LIN {X 0,Y 416.989,Z 554.741,A -85,B 0,C 180,E1 -10166.135,E2 -10166.135} C_VEL
LIN {X 0,Y 417.027,Z 556.75,A -85,B 0,C 180,E1 -10168.069,E2 -10168.069} C_VEL
LIN {X 0,Y 416.981,Z 557.414,A -85,B 0,C 180,E1 -10170,E2 -10170} C_VEL
LIN {X 0,Y 417.027,Z 556.748,A -85,B 0,C 180,E1 -10171.932,E2 -10171.932} C_VEL
LIN {X 0,Y 416.989,Z 554.738,A -85,B 0,C 180,E1 -10173.866,E2 -10173.866} C_VEL
LIN {X 0,Y 417.129,Z 551.337,A -85,B 0,C 180,E1 -10175.802,E2 -10175.802} C_VEL
LIN {X 0,Y 417.316,Z 546.442,A -85,B 0,C 180,E1 -10177.743,E2 -10177.743} C_VEL
LIN {X 0,Y 417.74,Z 539.91,A -85,B 0,C 180,E1 -10179.685,E2 -10179.685} C_VEL
LIN {X 0,Y 418.314,Z 532.641,A -85,B 0,C 180,E1 -10181.385,E2 -10181.385} C_VEL
LIN {X 0,Y 418.978,Z 524.176,A -85,B 0,C 180,E1 -10182.995,E2 -10182.995} C_VEL
LIN {X 0,Y 419.845,Z 514.188,A -85,B 0,C 180,E1 -10184.542,E2 -10184.542} C_VEL
LIN {X 0,Y 420.766,Z 503.727,A -85,B 0,C 180,E1 -10185.873,E2 -10185.873} C_VEL
LIN {X 0,Y 421.802,Z 492.183,A -85,B 0,C 180,E1 -10187.077,E2 -10187.077} C_VEL
LIN {X 0,Y 422.858,Z 479.374,A -85,B 0,C 180,E1 -10188.157,E2 -10188.157} C_VEL
LIN {X 0,Y 423.8,Z 466.334,A -85,B 0,C 180,E1 -10189.025,E2 -10189.025} C_VEL
LIN {X 0,Y 424.522,Z 452.931,A -85,B 0,C 180,E1 -10189.713,E2 -10189.713} C_VEL
LIN {X 0,Y 425.232,Z 438.211,A -85,B 0,C 180,E1 -10190.245,E2 -10190.245} C_VEL
LIN {X 0,Y 425.645,Z 423.401,A -85,B 0,C 180,E1 -10190.572,E2 -10190.572} C_VEL
LIN {X 0,Y 426.978,Z 321.763,A -85,B 0,C 180,E1 -10192.302,E2 -10192.302} C_VEL
LIN {X 0,Y 421.78,Z 294.783,A -85,B 0,C 180,E1 -10193.108,E2 -10193.108} C_VEL
LIN {X 0,Y 422.402,Z 285.458,A -85,B 0,C 180,E1 -10194.841,E2 -10194.841} C_VEL
LIN {X 0,Y 420.106,Z 273.797,A -85,B 0,C 180,E1 -10197.302,E2 -10197.302} C_VEL
LIN {X 0,Y 418.323,Z 266.179,A -85,B 0,C 180,E1 -10199.01,E2 -10199.01} C_VEL
LIN {X 0,Y 418.244,Z 266.011,A -85,B 0,C 180,E1 -10202.527,E2 -10202.527} C_VEL
LIN {X 0,Y 418.257,Z 266.012,A -85,B 0,C 180,E1 -10204.84,E2 -10204.84} C_VEL
LIN {X 0,Y 418.25,Z 266.009,A -85,B 0,C 180,E1 -10208.441,E2 -10208.441} C_VEL
LIN {X 0,Y 418.219,Z 265.999,A -85,B 0,C 180,E1 -10210.947,E2 -10210.947} C_VEL
LIN {X 0,Y 418.213,Z 266.013,A -85,B 0,C 180,E1 -10213.73,E2 -10213.73} C_VEL
LIN {X 0,Y 418.205,Z 266.016,A -85,B 0,C 180,E1 -10216.448,E2 -10216.448} C_VEL
LIN {X 0,Y 418.22,Z 266.007,A -85,B 0,C 180,E1 -10219.129,E2 -10219.129} C_VEL
LIN {X 0,Y 418.23,Z 266.013,A -85,B 0,C 180,E1 -10222.165,E2 -10222.165} C_VEL
LIN {X 0,Y 418.26,Z 265.977,A -85,B 0,C 180,E1 -10225.419,E2 -10225.419} C_VEL
LIN {X 0,Y 418.217,Z 266.013,A -85,B 0,C 180,E1 -10228.604,E2 -10228.604} C_VEL
LIN {X 0,Y 418.289,Z 266,A -85,B 0,C 180,E1 -10231.937,E2 -10231.937} C_VEL
LIN {X 0,Y 418.283,Z 266.004,A -85,B 0,C 180,E1 -10235.162,E2 -10235.162} C_VEL
LIN {X 0,Y 418.227,Z 266.008,A -85,B 0,C 180,E1 -10238.303,E2 -10238.303} C_VEL
LIN {X 0,Y 418.276,Z 266.007,A -85,B 0,C 180,E1 -10241.383,E2 -10241.383} C_VEL
LIN {X 0,Y 418.294,Z 266,A -85,B 0,C 180,E1 -10244.406,E2 -10244.406} C_VEL
LIN {X 0,Y 418.348,Z 265.999,A -85,B 0,C 180,E1 -10247.385,E2 -10247.385} C_VEL
LIN {X 0,Y 418.333,Z 265.992,A -85,B 0,C 180,E1 -10250.329,E2 -10250.329} C_VEL
LIN {X 0,Y 418.506,Z 265.977,A -85,B 0,C 180,E1 -10252.279,E2 -10252.279} C_VEL
LIN {X 0,Y 418.505,Z 265.972,A -85,B 0,C 180,E1 -10254.217,E2 -10254.217} C_VEL
LIN {X 0,Y 418.537,Z 265.973,A -85,B 0,C 180,E1 -10258.076,E2 -10258.076} C_VEL
LIN {X 0,Y 418.664,Z 265.956,A -85,B 0,C 180,E1 -10260,E2 -10260} C_VEL
LIN {X 0,Y 418.504,Z 265.964,A -85,B 0,C 180,E1 -10262.888,E2 -10262.888} C_VEL
LIN {X 0,Y 418.486,Z 265.979,A -85,B 0,C 180,E1 -10266.751,E2 -10266.751} C_VEL
LIN {X 0,Y 418.333,Z 265.994,A -85,B 0,C 180,E1 -10269.672,E2 -10269.672} C_VEL
LIN {X 0,Y 418.339,Z 266.001,A -85,B 0,C 180,E1 -10273.001,E2 -10273.001} C_VEL
LIN {X 0,Y 418.306,Z 265.999,A -85,B 0,C 180,E1 -10276.736,E2 -10276.736} C_VEL
LIN {X 0,Y 418.264,Z 266.001,A -85,B 0,C 180,E1 -10279.791,E2 -10279.791} C_VEL
LIN {X 0,Y 418.232,Z 266.01,A -85,B 0,C 180,E1 -10282.737,E2 -10282.737} C_VEL
LIN {X 0,Y 418.264,Z 265.998,A -85,B 0,C 180,E1 -10285.905,E2 -10285.905} C_VEL
LIN {X 0,Y 418.269,Z 266.009,A -85,B 0,C 180,E1 -10289.162,E2 -10289.162} C_VEL
LIN {X 0,Y 418.252,Z 265.98,A -85,B 0,C 180,E1 -10292.845,E2 -10292.845} C_VEL
LIN {X 0,Y 418.244,Z 266.004,A -85,B 0,C 180,E1 -10296.239,E2 -10296.239} C_VEL
LIN {X 0,Y 418.26,Z 266,A -85,B 0,C 180,E1 -10299.681,E2 -10299.681} C_VEL
LIN {X 0,Y 418.241,Z 265.99,A -85,B 0,C 180,E1 -10302.324,E2 -10302.324} C_VEL
LIN {X 0,Y 418.236,Z 266.012,A -85,B 0,C 180,E1 -10305.11,E2 -10305.11} C_VEL
LIN {X 0,Y 418.239,Z 265.993,A -85,B 0,C 180,E1 -10307.768,E2 -10307.768} C_VEL
LIN {X 0,Y 418.256,Z 266.011,A -85,B 0,C 180,E1 -10310.619,E2 -10310.619} C_VEL
LIN {X 0,Y 418.242,Z 266.011,A -85,B 0,C 180,E1 -10313.977,E2 -10313.977} C_VEL
LIN {X 0,Y 418.257,Z 266.011,A -85,B 0,C 180,E1 -10317.157,E2 -10317.157} C_VEL
LIN {X 0,Y 418.268,Z 265.996,A -85,B 0,C 180,E1 -10320.896,E2 -10320.896} C_VEL
LIN {X 0,Y 418.345,Z 266.202,A -85,B 0,C 180,E1 -10322.251,E2 -10322.251} C_VEL
LIN {X 0,Y 420.857,Z 277.948,A -85,B 0,C 180,E1 -10324.922,E2 -10324.922} C_VEL
LIN {X 0,Y 422.1,Z 284.986,A -85,B 0,C 180,E1 -10326.447,E2 -10326.447} C_VEL
LIN {X 0,Y 421.937,Z 287.927,A -85,B 0,C 180,E1 -10326.964,E2 -10326.964} C_VEL
LIN {X 0,Y 427.164,Z 313.752,A -85,B 0,C 180,E1 -10327.742,E2 -10327.742} C_VEL
LIN {X 0,Y 425.741,Z 409.801,A -85,B 0,C 180,E1 -10329.37,E2 -10329.37} C_VEL
LIN {X 0,Y 425.346,Z 427.971,A -85,B 0,C 180,E1 -10329.729,E2 -10329.729} C_VEL
LIN {X 0,Y 424.78,Z 442.274,A -85,B 0,C 180,E1 -10330.205,E2 -10330.205} C_VEL
LIN {X 0,Y 424.143,Z 455.506,A -85,B 0,C 180,E1 -10330.837,E2 -10330.837} C_VEL
LIN {X 0,Y 423.336,Z 467.967,A -85,B 0,C 180,E1 -10331.614,E2 -10331.614} C_VEL
LIN {X 0,Y 422.393,Z 480.205,A -85,B 0,C 180,E1 -10332.573,E2 -10332.573} C_VEL
LIN {X 0,Y 421.296,Z 492.545,A -85,B 0,C 180,E1 -10333.775,E2 -10333.775} C_VEL
LIN {X 0,Y 420.401,Z 502.683,A -85,B 0,C 180,E1 -10334.982,E2 -10334.982} C_VEL
LIN {X 0,Y 419.457,Z 512.747,A -85,B 0,C 180,E1 -10336.434,E2 -10336.434} C_VEL
LIN {X 0,Y 419.259,Z 516.218,A -85,B 0,C 180,E1 -10337.009,E2 -10337.009} C_VEL
LIN {X 0,Y 418.347,Z 519.856,A -85,B 0,C 180,E1 -10337.639,E2 -10337.639} C_VEL
LIN {X 0,Y 415.001,Z 525.435,A -85,B 0,C 180,E1 -10338.669,E2 -10338.669} C_VEL
LIN {X 0,Y 411.657,Z 530.499,A -85,B 0,C 180,E1 -10339.758,E2 -10339.758} C_VEL
LIN {X 0,Y 410.76,Z 533.265,A -85,B 0,C 180,E1 -10340.473,E2 -10340.473} C_VEL
LIN {X 0,Y 410.371,Z 538.623,A -85,B 0,C 180,E1 -10342.125,E2 -10342.125} C_VEL
LIN {X 0,Y 410.13,Z 543.523,A -85,B 0,C 180,E1 -10344.099,E2 -10344.099} C_VEL
LIN {X 0,Y 409.943,Z 546.935,A -85,B 0,C 180,E1 -10346.068,E2 -10346.068} C_VEL
LIN {X 0,Y 409.966,Z 548.961,A -85,B 0,C 180,E1 -10348.035,E2 -10348.035} C_VEL
LIN {X 0,Y 409.905,Z 549.659,A -85,B 0,C 180,E1 -10350,E2 -10350} C_VEL
LIN {X 0,Y 409.966,Z 549.033,A -85,B 0,C 180,E1 -10351.965,E2 -10351.965} C_VEL
LIN {X 0,Y 409.942,Z 547.071,A -85,B 0,C 180,E1 -10353.932,E2 -10353.932} C_VEL
LIN {X 0,Y 410.14,Z 543.725,A -85,B 0,C 180,E1 -10355.901,E2 -10355.901} C_VEL
LIN {X 0,Y 410.369,Z 538.899,A -85,B 0,C 180,E1 -10357.875,E2 -10357.875} C_VEL
LIN {X 0,Y 410.841,Z 532.438,A -85,B 0,C 180,E1 -10359.849,E2 -10359.849} C_VEL
LIN {X 0,Y 411.449,Z 525.242,A -85,B 0,C 180,E1 -10361.578,E2 -10361.578} C_VEL
LIN {X 0,Y 412.23,Z 516.795,A -85,B 0,C 180,E1 -10363.224,E2 -10363.224} C_VEL
LIN {X 0,Y 413.12,Z 506.993,A -85,B 0,C 180,E1 -10364.784,E2 -10364.784} C_VEL
LIN {X 0,Y 414.127,Z 496.637,A -85,B 0,C 180,E1 -10366.134,E2 -10366.134} C_VEL
LIN {X 0,Y 415.182,Z 485.209,A -85,B 0,C 180,E1 -10367.358,E2 -10367.358} C_VEL
LIN {X 0,Y 416.255,Z 472.542,A -85,B 0,C 180,E1 -10368.455,E2 -10368.455} C_VEL
LIN {X 0,Y 417.199,Z 459.111,A -85,B 0,C 180,E1 -10369.376,E2 -10369.376} C_VEL
LIN {X 0,Y 418.011,Z 445.27,A -85,B 0,C 180,E1 -10370.097,E2 -10370.097} C_VEL
LIN {X 0,Y 418.668,Z 431.435,A -85,B 0,C 180,E1 -10370.609,E2 -10370.609} C_VEL
LIN {X 0,Y 419.122,Z 417.109,A -85,B 0,C 180,E1 -10370.939,E2 -10370.939} C_VEL
LIN {X 0,Y 420.535,Z 313.798,A -85,B 0,C 180,E1 -10372.727,E2 -10372.727} C_VEL
LIN {X 0,Y 415.163,Z 287.798,A -85,B 0,C 180,E1 -10373.549,E2 -10373.549} C_VEL
LIN {X 0,Y 414.947,Z 284.257,A -85,B 0,C 180,E1 -10374.25,E2 -10374.25} C_VEL
LIN {X 0,Y 412.295,Z 271.516,A -85,B 0,C 180,E1 -10377.127,E2 -10377.127} C_VEL
LIN {X 0,Y 411.27,Z 266.99,A -85,B 0,C 180,E1 -10378.237,E2 -10378.237} C_VEL
LIN {X 0,Y 411.164,Z 266.891,A -85,B 0,C 180,E1 -10381.997,E2 -10381.997} C_VEL
LIN {X 0,Y 411.209,Z 266.884,A -85,B 0,C 180,E1 -10384.878,E2 -10384.878} C_VEL
LIN {X 0,Y 411.204,Z 266.88,A -85,B 0,C 180,E1 -10388.168,E2 -10388.168} C_VEL
LIN {X 0,Y 411.162,Z 266.887,A -85,B 0,C 180,E1 -10391.228,E2 -10391.228} C_VEL
LIN {X 0,Y 411.176,Z 266.889,A -85,B 0,C 180,E1 -10394.489,E2 -10394.489} C_VEL
LIN {X 0,Y 411.194,Z 266.865,A -85,B 0,C 180,E1 -10398.196,E2 -10398.196} C_VEL
LIN {X 0,Y 411.226,Z 266.879,A -85,B 0,C 180,E1 -10400.777,E2 -10400.777} C_VEL
LIN {X 0,Y 411.194,Z 266.884,A -85,B 0,C 180,E1 -10404.471,E2 -10404.471} C_VEL
LIN {X 0,Y 411.201,Z 266.857,A -85,B 0,C 180,E1 -10406.873,E2 -10406.873} C_VEL
LIN {X 0,Y 411.235,Z 266.884,A -85,B 0,C 180,E1 -10410.642,E2 -10410.642} C_VEL
LIN {X 0,Y 411.231,Z 266.875,A -85,B 0,C 180,E1 -10413.618,E2 -10413.618} C_VEL
LIN {X 0,Y 411.196,Z 266.893,A -85,B 0,C 180,E1 -10416.852,E2 -10416.852} C_VEL
LIN {X 0,Y 411.207,Z 266.879,A -85,B 0,C 180,E1 -10420.05,E2 -10420.05} C_VEL
LIN {X 0,Y 411.255,Z 266.879,A -85,B 0,C 180,E1 -10423.131,E2 -10423.131} C_VEL
LIN {X 0,Y 411.297,Z 266.876,A -85,B 0,C 180,E1 -10426.896,E2 -10426.896} C_VEL
LIN {X 0,Y 411.286,Z 266.873,A -85,B 0,C 180,E1 -10430.161,E2 -10430.161} C_VEL
LIN {X 0,Y 411.453,Z 266.856,A -85,B 0,C 180,E1 -10433.133,E2 -10433.133} C_VEL
LIN {X 0,Y 411.305,Z 266.873,A -85,B 0,C 180,E1 -10435.099,E2 -10435.099} C_VEL
LIN {X 0,Y 411.506,Z 266.835,A -85,B 0,C 180,E1 -10438.042,E2 -10438.042} C_VEL
LIN {X 0,Y 411.635,Z 266.831,A -85,B 0,C 180,E1 -10440,E2 -10440} C_VEL
LIN {X 0,Y 411.458,Z 266.846,A -85,B 0,C 180,E1 -10442.937,E2 -10442.937} C_VEL
LIN {X 0,Y 411.452,Z 266.857,A -85,B 0,C 180,E1 -10446.867,E2 -10446.867} C_VEL
LIN {X 0,Y 411.346,Z 266.863,A -85,B 0,C 180,E1 -10448.845,E2 -10448.845} C_VEL
LIN {X 0,Y 411.275,Z 266.873,A -85,B 0,C 180,E1 -10451.833,E2 -10451.833} C_VEL
LIN {X 0,Y 411.252,Z 266.877,A -85,B 0,C 180,E1 -10454.853,E2 -10454.853} C_VEL
LIN {X 0,Y 411.244,Z 266.878,A -85,B 0,C 180,E1 -10457.915,E2 -10457.915} C_VEL
LIN {X 0,Y 411.188,Z 266.883,A -85,B 0,C 180,E1 -10461.034,E2 -10461.034} C_VEL
LIN {X 0,Y 411.22,Z 266.889,A -85,B 0,C 180,E1 -10464.216,E2 -10464.216} C_VEL
LIN {X 0,Y 411.253,Z 266.873,A -85,B 0,C 180,E1 -10467.478,E2 -10467.478} C_VEL
LIN {X 0,Y 411.194,Z 266.886,A -85,B 0,C 180,E1 -10470.847,E2 -10470.847} C_VEL
LIN {X 0,Y 411.2,Z 266.856,A -85,B 0,C 180,E1 -10474.334,E2 -10474.334} C_VEL
LIN {X 0,Y 411.195,Z 266.892,A -85,B 0,C 180,E1 -10477.974,E2 -10477.974} C_VEL
LIN {X 0,Y 411.178,Z 266.885,A -85,B 0,C 180,E1 -10480.505,E2 -10480.505} C_VEL
LIN {X 0,Y 411.168,Z 266.892,A -85,B 0,C 180,E1 -10483.134,E2 -10483.134} C_VEL
LIN {X 0,Y 411.223,Z 266.887,A -85,B 0,C 180,E1 -10485.873,E2 -10485.873} C_VEL
LIN {X 0,Y 411.206,Z 266.871,A -85,B 0,C 180,E1 -10488.765,E2 -10488.765} C_VEL
LIN {X 0,Y 411.201,Z 266.881,A -85,B 0,C 180,E1 -10492.028,E2 -10492.028} C_VEL
LIN {X 0,Y 411.203,Z 266.883,A -85,B 0,C 180,E1 -10495.667,E2 -10495.667} C_VEL
LIN {X 0,Y 411.187,Z 266.868,A -85,B 0,C 180,E1 -10499.153,E2 -10499.153} C_VEL
LIN {X 0,Y 411.234,Z 267.106,A -85,B 0,C 180,E1 -10500.644,E2 -10500.644} C_VEL
LIN {X 0,Y 413.937,Z 278.724,A -85,B 0,C 180,E1 -10503.262,E2 -10503.262} C_VEL
LIN {X 0,Y 415.499,Z 286.781,A -85,B 0,C 180,E1 -10504.985,E2 -10504.985} C_VEL
LIN {X 0,Y 414.986,Z 294.728,A -85,B 0,C 180,E1 -10506.484,E2 -10506.484} C_VEL
LIN {X 0,Y 420.238,Z 321.769,A -85,B 0,C 180,E1 -10507.314,E2 -10507.314} C_VEL
LIN {X 0,Y 420.434,Z 325.335,A -85,B 0,C 180,E1 -10507.39,E2 -10507.39} C_VEL
LIN {X 0,Y 418.966,Z 425.486,A -85,B 0,C 180,E1 -10509.118,E2 -10509.118} C_VEL
LIN {X 0,Y 418.466,Z 440.252,A -85,B 0,C 180,E1 -10509.477,E2 -10509.477} C_VEL
LIN {X 0,Y 417.775,Z 454.321,A -85,B 0,C 180,E1 -10510.02,E2 -10510.02} C_VEL
LIN {X 0,Y 416.956,Z 467.449,A -85,B 0,C 180,E1 -10510.719,E2 -10510.719} C_VEL
LIN {X 0,Y 415.953,Z 480.97,A -85,B 0,C 180,E1 -10511.658,E2 -10511.658} C_VEL
LIN {X 0,Y 414.891,Z 493.475,A -85,B 0,C 180,E1 -10512.757,E2 -10512.757} C_VEL
LIN {X 0,Y 413.806,Z 504.781,A -85,B 0,C 180,E1 -10513.98,E2 -10513.98} C_VEL
LIN {X 0,Y 412.771,Z 515.853,A -85,B 0,C 180,E1 -10515.455,E2 -10515.455} C_VEL
LIN {X 0,Y 411.989,Z 524.629,A -85,B 0,C 180,E1 -10516.871,E2 -10516.871} C_VEL
LIN {X 0,Y 411.33,Z 532.6,A -85,B 0,C 180,E1 -10518.419,E2 -10518.419} C_VEL
LIN {X 0,Y 410.704,Z 539.864,A -85,B 0,C 180,E1 -10520.147,E2 -10520.147} C_VEL
LIN {X 0,Y 410.258,Z 546.393,A -85,B 0,C 180,E1 -10522.123,E2 -10522.123} C_VEL
LIN {X 0,Y 410.046,Z 551.279,A -85,B 0,C 180,E1 -10524.098,E2 -10524.098} C_VEL
LIN {X 0,Y 409.908,Z 554.675,A -85,B 0,C 180,E1 -10526.068,E2 -10526.068} C_VEL
LIN {X 0,Y 409.923,Z 556.684,A -85,B 0,C 180,E1 -10528.035,E2 -10528.035} C_VEL
LIN {X 0,Y 409.904,Z 557.348,A -85,B 0,C 180,E1 -10530,E2 -10530} C_VEL
LIN {X 0,Y 409.923,Z 556.681,A -85,B 0,C 180,E1 -10531.965,E2 -10531.965} C_VEL
LIN {X 0,Y 409.908,Z 554.671,A -85,B 0,C 180,E1 -10533.932,E2 -10533.932} C_VEL
LIN {X 0,Y 410.053,Z 551.27,A -85,B 0,C 180,E1 -10535.902,E2 -10535.902} C_VEL
LIN {X 0,Y 410.258,Z 546.374,A -85,B 0,C 180,E1 -10537.877,E2 -10537.877} C_VEL
LIN {X 0,Y 410.709,Z 539.842,A -85,B 0,C 180,E1 -10539.853,E2 -10539.853} C_VEL
LIN {X 0,Y 411.326,Z 532.573,A -85,B 0,C 180,E1 -10541.581,E2 -10541.581} C_VEL
LIN {X 0,Y 411.964,Z 524.669,A -85,B 0,C 180,E1 -10543.116,E2 -10543.116} C_VEL
LIN {X 0,Y 412.785,Z 515.811,A -85,B 0,C 180,E1 -10544.544,E2 -10544.544} C_VEL
LIN {X 0,Y 413.804,Z 504.724,A -85,B 0,C 180,E1 -10546.021,E2 -10546.021} C_VEL
LIN {X 0,Y 414.898,Z 493.405,A -85,B 0,C 180,E1 -10547.243,E2 -10547.243} C_VEL
LIN {X 0,Y 415.971,Z 480.886,A -85,B 0,C 180,E1 -10548.341,E2 -10548.341} C_VEL
LIN {X 0,Y 416.991,Z 467.413,A -85,B 0,C 180,E1 -10549.274,E2 -10549.274} C_VEL
LIN {X 0,Y 417.771,Z 454.158,A -85,B 0,C 180,E1 -10549.981,E2 -10549.981} C_VEL
LIN {X 0,Y 418.48,Z 440.032,A -85,B 0,C 180,E1 -10550.522,E2 -10550.522} C_VEL
LIN {X 0,Y 418.917,Z 426.639,A -85,B 0,C 180,E1 -10550.853,E2 -10550.853} C_VEL
LIN {X 0,Y 420.457,Z 323.733,A -85,B 0,C 180,E1 -10552.63,E2 -10552.63} C_VEL
LIN {X 0,Y 417.351,Z 306.745,A -85,B 0,C 180,E1 -10553.118,E2 -10553.118} C_VEL
LIN {X 0,Y 414.961,Z 294.802,A -85,B 0,C 180,E1 -10553.502,E2 -10553.502} C_VEL
LIN {X 0,Y 415.48,Z 286.73,A -85,B 0,C 180,E1 -10555.016,E2 -10555.016} C_VEL
LIN {X 0,Y 413.367,Z 275.981,A -85,B 0,C 180,E1 -10557.325,E2 -10557.325} C_VEL
LIN {X 0,Y 411.232,Z 267.075,A -85,B 0,C 180,E1 -10559.355,E2 -10559.355} C_VEL
LIN {X 0,Y 411.164,Z 266.894,A -85,B 0,C 180,E1 -10561.997,E2 -10561.997} C_VEL
LIN {X 0,Y 411.208,Z 266.891,A -85,B 0,C 180,E1 -10564.878,E2 -10564.878} C_VEL
LIN {X 0,Y 411.201,Z 266.883,A -85,B 0,C 180,E1 -10568.168,E2 -10568.168} C_VEL
LIN {X 0,Y 411.161,Z 266.876,A -85,B 0,C 180,E1 -10571.228,E2 -10571.228} C_VEL
LIN {X 0,Y 411.176,Z 266.893,A -85,B 0,C 180,E1 -10574.489,E2 -10574.489} C_VEL
LIN {X 0,Y 411.173,Z 266.893,A -85,B 0,C 180,E1 -10578.194,E2 -10578.194} C_VEL
LIN {X 0,Y 411.219,Z 266.886,A -85,B 0,C 180,E1 -10580.776,E2 -10580.776} C_VEL
LIN {X 0,Y 411.194,Z 266.862,A -85,B 0,C 180,E1 -10584.471,E2 -10584.471} C_VEL
LIN {X 0,Y 411.166,Z 266.883,A -85,B 0,C 180,E1 -10588.003,E2 -10588.003} C_VEL
LIN {X 0,Y 411.218,Z 266.884,A -85,B 0,C 180,E1 -10591.41,E2 -10591.41} C_VEL
LIN {X 0,Y 411.23,Z 266.883,A -85,B 0,C 180,E1 -10594.707,E2 -10594.707} C_VEL
LIN {X 0,Y 411.199,Z 266.881,A -85,B 0,C 180,E1 -10597.913,E2 -10597.913} C_VEL
LIN {X 0,Y 411.217,Z 266.884,A -85,B 0,C 180,E1 -10601.051,E2 -10601.051} C_VEL
LIN {X 0,Y 411.247,Z 266.876,A -85,B 0,C 180,E1 -10604.131,E2 -10604.131} C_VEL
LIN {X 0,Y 411.295,Z 266.876,A -85,B 0,C 180,E1 -10607.165,E2 -10607.165} C_VEL
LIN {X 0,Y 411.285,Z 266.87,A -85,B 0,C 180,E1 -10610.161,E2 -10610.161} C_VEL
LIN {X 0,Y 411.475,Z 266.854,A -85,B 0,C 180,E1 -10612.147,E2 -10612.147} C_VEL
LIN {X 0,Y 411.467,Z 266.85,A -85,B 0,C 180,E1 -10614.118,E2 -10614.118} C_VEL
LIN {X 0,Y 411.506,Z 266.849,A -85,B 0,C 180,E1 -10618.043,E2 -10618.043} C_VEL
LIN {X 0,Y 411.634,Z 266.832,A -85,B 0,C 180,E1 -10620,E2 -10620} C_VEL
LIN {X 0,Y 411.459,Z 266.841,A -85,B 0,C 180,E1 -10622.937,E2 -10622.937} C_VEL
LIN {X 0,Y 411.449,Z 266.856,A -85,B 0,C 180,E1 -10626.867,E2 -10626.867} C_VEL
LIN {X 0,Y 411.285,Z 266.873,A -85,B 0,C 180,E1 -10629.839,E2 -10629.839} C_VEL
LIN {X 0,Y 411.298,Z 266.877,A -85,B 0,C 180,E1 -10633.105,E2 -10633.105} C_VEL
LIN {X 0,Y 411.256,Z 266.878,A -85,B 0,C 180,E1 -10636.869,E2 -10636.869} C_VEL
LIN {X 0,Y 411.224,Z 266.877,A -85,B 0,C 180,E1 -10639.987,E2 -10639.987} C_VEL
LIN {X 0,Y 411.197,Z 266.892,A -85,B 0,C 180,E1 -10643.148,E2 -10643.148} C_VEL
LIN {X 0,Y 411.232,Z 266.874,A -85,B 0,C 180,E1 -10646.381,E2 -10646.381} C_VEL
LIN {X 0,Y 411.205,Z 266.884,A -85,B 0,C 180,E1 -10649.712,E2 -10649.712} C_VEL
LIN {X 0,Y 411.201,Z 266.855,A -85,B 0,C 180,E1 -10653.156,E2 -10653.156} C_VEL
LIN {X 0,Y 411.191,Z 266.885,A -85,B 0,C 180,E1 -10656.554,E2 -10656.554} C_VEL
LIN {X 0,Y 411.222,Z 266.876,A -85,B 0,C 180,E1 -10659.731,E2 -10659.731} C_VEL
LIN {X 0,Y 411.174,Z 266.882,A -85,B 0,C 180,E1 -10663.134,E2 -10663.134} C_VEL
LIN {X 0,Y 411.17,Z 266.89,A -85,B 0,C 180,E1 -10665.881,E2 -10665.881} C_VEL
LIN {X 0,Y 411.163,Z 266.884,A -85,B 0,C 180,E1 -10668.772,E2 -10668.772} C_VEL
LIN {X 0,Y 411.205,Z 266.88,A -85,B 0,C 180,E1 -10671.832,E2 -10671.832} C_VEL
LIN {X 0,Y 411.21,Z 266.883,A -85,B 0,C 180,E1 -10675.122,E2 -10675.122} C_VEL
LIN {X 0,Y 411.165,Z 266.892,A -85,B 0,C 180,E1 -10678.003,E2 -10678.003} C_VEL
LIN {X 0,Y 411.254,Z 266.886,A -85,B 0,C 180,E1 -10681.762,E2 -10681.762} C_VEL
LIN {X 0,Y 411.348,Z 267.271,A -85,B 0,C 180,E1 -10681.977,E2 -10681.977} C_VEL
LIN {X 0,Y 414.076,Z 279.964,A -85,B 0,C 180,E1 -10684.893,E2 -10684.893} C_VEL
LIN {X 0,Y 415.101,Z 285.424,A -85,B 0,C 180,E1 -10686.102,E2 -10686.102} C_VEL
LIN {X 0,Y 415.145,Z 287.898,A -85,B 0,C 180,E1 -10686.557,E2 -10686.557} C_VEL
LIN {X 0,Y 420.509,Z 313.956,A -85,B 0,C 180,E1 -10687.373,E2 -10687.373} C_VEL
LIN {X 0,Y 419.264,Z 404.529,A -85,B 0,C 180,E1 -10688.94,E2 -10688.94} C_VEL
LIN {X 0,Y 418.762,Z 426.915,A -85,B 0,C 180,E1 -10689.364,E2 -10689.364} C_VEL
LIN {X 0,Y 418.159,Z 441.591,A -85,B 0,C 180,E1 -10689.846,E2 -10689.846} C_VEL
LIN {X 0,Y 417.44,Z 455.806,A -85,B 0,C 180,E1 -10690.53,E2 -10690.53} C_VEL
LIN {X 0,Y 416.477,Z 469.76,A -85,B 0,C 180,E1 -10691.427,E2 -10691.427} C_VEL
LIN {X 0,Y 415.506,Z 481.646,A -85,B 0,C 180,E1 -10692.402,E2 -10692.402} C_VEL
LIN {X 0,Y 414.359,Z 493.683,A -85,B 0,C 180,E1 -10693.622,E2 -10693.622} C_VEL
LIN {X 0,Y 413.338,Z 504.533,A -85,B 0,C 180,E1 -10694.972,E2 -10694.972} C_VEL
LIN {X 0,Y 412.396,Z 514.185,A -85,B 0,C 180,E1 -10696.429,E2 -10696.429} C_VEL
LIN {X 0,Y 411.768,Z 522.397,A -85,B 0,C 180,E1 -10697.932,E2 -10697.932} C_VEL
LIN {X 0,Y 411.055,Z 530.153,A -85,B 0,C 180,E1 -10699.658,E2 -10699.658} C_VEL
LIN {X 0,Y 410.76,Z 533.265,A -85,B 0,C 180,E1 -10700.473,E2 -10700.473} C_VEL
LIN {X 0,Y 409.914,Z 535.864,A -85,B 0,C 180,E1 -10701.205,E2 -10701.205} C_VEL
LIN {X 0,Y 406.799,Z 539.678,A -85,B 0,C 180,E1 -10702.415,E2 -10702.415} C_VEL
LIN {X 0,Y 404.229,Z 542.314,A -85,B 0,C 180,E1 -10703.416,E2 -10703.416} C_VEL
LIN {X 0,Y 403.039,Z 544.309,A -85,B 0,C 180,E1 -10704.342,E2 -10704.342} C_VEL
LIN {X 0,Y 403.008,Z 544.497,A -85,B 0,C 180,E1 -10704.478,E2 -10704.478} C_VEL
LIN {X 0,Y 402.866,Z 547.002,A -85,B 0,C 180,E1 -10705.999,E2 -10705.999} C_VEL
LIN {X 0,Y 402.864,Z 549.028,A -85,B 0,C 180,E1 -10708.001,E2 -10708.001} C_VEL
LIN {X 0,Y 402.831,Z 549.725,A -85,B 0,C 180,E1 -10710,E2 -10710} C_VEL
LIN {X 0,Y 402.864,Z 549.099,A -85,B 0,C 180,E1 -10711.999,E2 -10711.999} C_VEL
LIN {X 0,Y 402.865,Z 547.137,A -85,B 0,C 180,E1 -10714.001,E2 -10714.001} C_VEL
LIN {X 0,Y 403.071,Z 543.791,A -85,B 0,C 180,E1 -10716.005,E2 -10716.005} C_VEL
LIN {X 0,Y 403.309,Z 538.965,A -85,B 0,C 180,E1 -10718.013,E2 -10718.013} C_VEL
LIN {X 0,Y 403.828,Z 532.503,A -85,B 0,C 180,E1 -10720.022,E2 -10720.022} C_VEL
LIN {X 0,Y 404.481,Z 525.307,A -85,B 0,C 180,E1 -10721.78,E2 -10721.78} C_VEL
LIN {X 0,Y 405.242,Z 517.343,A -85,B 0,C 180,E1 -10723.364,E2 -10723.364} C_VEL
LIN {X 0,Y 406.041,Z 508.713,A -85,B 0,C 180,E1 -10724.791,E2 -10724.791} C_VEL
LIN {X 0,Y 407.187,Z 497.744,A -85,B 0,C 180,E1 -10726.288,E2 -10726.288} C_VEL
LIN {X 0,Y 408.307,Z 486.559,A -85,B 0,C 180,E1 -10727.53,E2 -10727.53} C_VEL
LIN {X 0,Y 409.384,Z 474.183,A -85,B 0,C 180,E1 -10728.647,E2 -10728.647} C_VEL
LIN {X 0,Y 410.397,Z 461.476,A -85,B 0,C 180,E1 -10729.559,E2 -10729.559} C_VEL
LIN {X 0,Y 411.231,Z 447.927,A -85,B 0,C 180,E1 -10730.312,E2 -10730.312} C_VEL
LIN {X 0,Y 411.919,Z 433.323,A -85,B 0,C 180,E1 -10730.897,E2 -10730.897} C_VEL
LIN {X 0,Y 412.376,Z 420.297,A -85,B 0,C 180,E1 -10731.232,E2 -10731.232} C_VEL
LIN {X 0,Y 414.044,Z 315.675,A -85,B 0,C 180,E1 -10733.07,E2 -10733.07} C_VEL
LIN {X 0,Y 408.583,Z 289.014,A -85,B 0,C 180,E1 -10733.903,E2 -10733.903} C_VEL
LIN {X 0,Y 408.292,Z 287.44,A -85,B 0,C 180,E1 -10734.029,E2 -10734.029} C_VEL
LIN {X 0,Y 405.906,Z 275.398,A -85,B 0,C 180,E1 -10736.754,E2 -10736.754} C_VEL
LIN {X 0,Y 404.201,Z 267.926,A -85,B 0,C 180,E1 -10738.564,E2 -10738.564} C_VEL
LIN {X 0,Y 404.138,Z 267.764,A -85,B 0,C 180,E1 -10741.557,E2 -10741.557} C_VEL
LIN {X 0,Y 404.183,Z 267.76,A -85,B 0,C 180,E1 -10745.015,E2 -10745.015} C_VEL
LIN {X 0,Y 404.155,Z 267.761,A -85,B 0,C 180,E1 -10748.756,E2 -10748.756} C_VEL
LIN {X 0,Y 404.121,Z 267.757,A -85,B 0,C 180,E1 -10751.599,E2 -10751.599} C_VEL
LIN {X 0,Y 404.145,Z 267.765,A -85,B 0,C 180,E1 -10754.522,E2 -10754.522} C_VEL
LIN {X 0,Y 404.141,Z 267.752,A -85,B 0,C 180,E1 -10757.296,E2 -10757.296} C_VEL
LIN {X 0,Y 404.164,Z 267.753,A -85,B 0,C 180,E1 -10759.955,E2 -10759.955} C_VEL
LIN {X 0,Y 404.136,Z 267.772,A -85,B 0,C 180,E1 -10763.123,E2 -10763.123} C_VEL
LIN {X 0,Y 404.139,Z 267.737,A -85,B 0,C 180,E1 -10766.187,E2 -10766.187} C_VEL
LIN {X 0,Y 404.147,Z 267.765,A -85,B 0,C 180,E1 -10769.715,E2 -10769.715} C_VEL
LIN {X 0,Y 404.189,Z 267.756,A -85,B 0,C 180,E1 -10773.122,E2 -10773.122} C_VEL
LIN {X 0,Y 404.171,Z 267.766,A -85,B 0,C 180,E1 -10775.334,E2 -10775.334} C_VEL
LIN {X 0,Y 404.131,Z 267.763,A -85,B 0,C 180,E1 -10778.58,E2 -10778.58} C_VEL
LIN {X 0,Y 404.203,Z 267.758,A -85,B 0,C 180,E1 -10781.761,E2 -10781.761} C_VEL
LIN {X 0,Y 404.198,Z 267.751,A -85,B 0,C 180,E1 -10784.882,E2 -10784.882} C_VEL
LIN {X 0,Y 404.249,Z 267.752,A -85,B 0,C 180,E1 -10787.958,E2 -10787.958} C_VEL
LIN {X 0,Y 404.398,Z 267.725,A -85,B 0,C 180,E1 -10792.127,E2 -10792.127} C_VEL
LIN {X 0,Y 404.417,Z 267.732,A -85,B 0,C 180,E1 -10794.015,E2 -10794.015} C_VEL
LIN {X 0,Y 404.475,Z 267.711,A -85,B 0,C 180,E1 -10798.008,E2 -10798.008} C_VEL
LIN {X 0,Y 404.605,Z 267.707,A -85,B 0,C 180,E1 -10800,E2 -10800} C_VEL
LIN {X 0,Y 404.415,Z 267.723,A -85,B 0,C 180,E1 -10802.988,E2 -10802.988} C_VEL
LIN {X 0,Y 404.403,Z 267.734,A -85,B 0,C 180,E1 -10806.987,E2 -10806.987} C_VEL
LIN {X 0,Y 404.25,Z 267.744,A -85,B 0,C 180,E1 -10810.012,E2 -10810.012} C_VEL
LIN {X 0,Y 404.258,Z 267.751,A -85,B 0,C 180,E1 -10813.212,E2 -10813.212} C_VEL
LIN {X 0,Y 404.208,Z 267.751,A -85,B 0,C 180,E1 -10817.007,E2 -10817.007} C_VEL
LIN {X 0,Y 404.156,Z 267.764,A -85,B 0,C 180,E1 -10820.352,E2 -10820.352} C_VEL
LIN {X 0,Y 404.162,Z 267.76,A -85,B 0,C 180,E1 -10823.575,E2 -10823.575} C_VEL
LIN {X 0,Y 404.177,Z 267.765,A -85,B 0,C 180,E1 -10825.767,E2 -10825.767} C_VEL
LIN {X 0,Y 404.191,Z 267.755,A -85,B 0,C 180,E1 -10828,E2 -10828} C_VEL
LIN {X 0,Y 404.14,Z 267.764,A -85,B 0,C 180,E1 -10831.56,E2 -10831.56} C_VEL
LIN {X 0,Y 404.179,Z 267.732,A -85,B 0,C 180,E1 -10835.017,E2 -10835.017} C_VEL
LIN {X 0,Y 404.154,Z 267.765,A -85,B 0,C 180,E1 -10838.757,E2 -10838.757} C_VEL
LIN {X 0,Y 404.118,Z 267.769,A -85,B 0,C 180,E1 -10841.6,E2 -10841.6} C_VEL
LIN {X 0,Y 404.149,Z 267.764,A -85,B 0,C 180,E1 -10844.524,E2 -10844.524} C_VEL
LIN {X 0,Y 404.203,Z 267.75,A -85,B 0,C 180,E1 -10847.306,E2 -10847.306} C_VEL
LIN {X 0,Y 404.165,Z 267.762,A -85,B 0,C 180,E1 -10849.956,E2 -10849.956} C_VEL
LIN {X 0,Y 404.137,Z 267.756,A -85,B 0,C 180,E1 -10853.125,E2 -10853.125} C_VEL
LIN {X 0,Y 404.142,Z 267.758,A -85,B 0,C 180,E1 -10856.188,E2 -10856.188} C_VEL
LIN {X 0,Y 404.144,Z 267.737,A -85,B 0,C 180,E1 -10859.716,E2 -10859.716} C_VEL
LIN {X 0,Y 404.208,Z 268.03,A -85,B 0,C 180,E1 -10860.297,E2 -10860.297} C_VEL
LIN {X 0,Y 407.033,Z 280.003,A -85,B 0,C 180,E1 -10863.049,E2 -10863.049} C_VEL
LIN {X 0,Y 408.589,Z 288.056,A -85,B 0,C 180,E1 -10864.805,E2 -10864.805} C_VEL
LIN {X 0,Y 408.187,Z 294.523,A -85,B 0,C 180,E1 -10866.055,E2 -10866.055} C_VEL
LIN {X 0,Y 409.76,Z 302.409,A -85,B 0,C 180,E1 -10866.339,E2 -10866.339} C_VEL
LIN {X 0,Y 413.861,Z 323.843,A -85,B 0,C 180,E1 -10866.984,E2 -10866.984} C_VEL
LIN {X 0,Y 412.438,Z 420.108,A -85,B 0,C 180,E1 -10868.673,E2 -10868.673} C_VEL
LIN {X 0,Y 412.024,Z 436.077,A -85,B 0,C 180,E1 -10869.011,E2 -10869.011} C_VEL
LIN {X 0,Y 411.339,Z 450.151,A -85,B 0,C 180,E1 -10869.498,E2 -10869.498} C_VEL
LIN {X 0,Y 410.549,Z 463.663,A -85,B 0,C 180,E1 -10870.167,E2 -10870.167} C_VEL
LIN {X 0,Y 409.665,Z 476.096,A -85,B 0,C 180,E1 -10870.977,E2 -10870.977} C_VEL
LIN {X 0,Y 408.616,Z 488.214,A -85,B 0,C 180,E1 -10871.966,E2 -10871.966} C_VEL
LIN {X 0,Y 407.367,Z 500.44,A -85,B 0,C 180,E1 -10873.204,E2 -10873.204} C_VEL
LIN {X 0,Y 406.381,Z 510.533,A -85,B 0,C 180,E1 -10874.452,E2 -10874.452} C_VEL
LIN {X 0,Y 405.409,Z 520.567,A -85,B 0,C 180,E1 -10875.955,E2 -10875.955} C_VEL
LIN {X 0,Y 404.696,Z 528.9,A -85,B 0,C 180,E1 -10877.463,E2 -10877.463} C_VEL
LIN {X 0,Y 403.871,Z 536.865,A -85,B 0,C 180,E1 -10879.219,E2 -10879.219} C_VEL
LIN {X 0,Y 403.408,Z 543.279,A -85,B 0,C 180,E1 -10880.979,E2 -10880.979} C_VEL
LIN {X 0,Y 403.072,Z 548.965,A -85,B 0,C 180,E1 -10882.99,E2 -10882.99} C_VEL
LIN {X 0,Y 402.91,Z 553.089,A -85,B 0,C 180,E1 -10884.997,E2 -10884.997} C_VEL
LIN {X 0,Y 402.779,Z 555.782,A -85,B 0,C 180,E1 -10887,E2 -10887} C_VEL
LIN {X 0,Y 402.843,Z 557.116,A -85,B 0,C 180,E1 -10889,E2 -10889} C_VEL
LIN {X 0,Y 402.843,Z 557.115,A -85,B 0,C 180,E1 -10891,E2 -10891} C_VEL
LIN {X 0,Y 402.779,Z 555.778,A -85,B 0,C 180,E1 -10893.001,E2 -10893.001} C_VEL
LIN {X 0,Y 402.913,Z 553.082,A -85,B 0,C 180,E1 -10895.003,E2 -10895.003} C_VEL
LIN {X 0,Y 403.072,Z 548.949,A -85,B 0,C 180,E1 -10897.01,E2 -10897.01} C_VEL
LIN {X 0,Y 403.412,Z 543.256,A -85,B 0,C 180,E1 -10899.021,E2 -10899.021} C_VEL
LIN {X 0,Y 403.871,Z 536.838,A -85,B 0,C 180,E1 -10900.781,E2 -10900.781} C_VEL
LIN {X 0,Y 404.699,Z 528.866,A -85,B 0,C 180,E1 -10902.537,E2 -10902.537} C_VEL
LIN {X 0,Y 405.406,Z 520.524,A -85,B 0,C 180,E1 -10904.046,E2 -10904.046} C_VEL
LIN {X 0,Y 406.385,Z 510.482,A -85,B 0,C 180,E1 -10905.548,E2 -10905.548} C_VEL
LIN {X 0,Y 407.478,Z 499.278,A -85,B 0,C 180,E1 -10906.921,E2 -10906.921} C_VEL
LIN {X 0,Y 408.759,Z 486.706,A -85,B 0,C 180,E1 -10908.157,E2 -10908.157} C_VEL
LIN {X 0,Y 409.794,Z 473.819,A -85,B 0,C 180,E1 -10909.176,E2 -10909.176} C_VEL
LIN {X 0,Y 410.735,Z 460.252,A -85,B 0,C 180,E1 -10910.011,E2 -10910.011} C_VEL
LIN {X 0,Y 411.593,Z 446.136,A -85,B 0,C 180,E1 -10910.653,E2 -10910.653} C_VEL
LIN {X 0,Y 412.133,Z 432.362,A -85,B 0,C 180,E1 -10911.082,E2 -10911.082} C_VEL
LIN {X 0,Y 413.661,Z 339.907,A -85,B 0,C 180,E1 -10912.723,E2 -10912.723} C_VEL
LIN {X 0,Y 413.843,Z 323.748,A -85,B 0,C 180,E1 -10913.011,E2 -10913.011} C_VEL
LIN {X 0,Y 408.209,Z 295.032,A -85,B 0,C 180,E1 -10913.898,E2 -10913.898} C_VEL
LIN {X 0,Y 408.257,Z 293.203,A -85,B 0,C 180,E1 -10914.164,E2 -10914.164} C_VEL
LIN {X 0,Y 408.579,Z 288.003,A -85,B 0,C 180,E1 -10915.196,E2 -10915.196} C_VEL
LIN {X 0,Y 405.946,Z 275.277,A -85,B 0,C 180,E1 -10918,E2 -10918} C_VEL
LIN {X 0,Y 404.209,Z 267.984,A -85,B 0,C 180,E1 -10919.703,E2 -10919.703} C_VEL
LIN {X 0,Y 404.144,Z 267.738,A -85,B 0,C 180,E1 -10920.285,E2 -10920.285} C_VEL
LIN {X 0,Y 404.143,Z 267.758,A -85,B 0,C 180,E1 -10923.812,E2 -10923.812} C_VEL
LIN {X 0,Y 404.133,Z 267.757,A -85,B 0,C 180,E1 -10926.874,E2 -10926.874} C_VEL
LIN {X 0,Y 404.144,Z 267.763,A -85,B 0,C 180,E1 -10930.079,E2 -10930.079} C_VEL
LIN {X 0,Y 404.153,Z 267.764,A -85,B 0,C 180,E1 -10933.084,E2 -10933.084} C_VEL
LIN {X 0,Y 404.145,Z 267.764,A -85,B 0,C 180,E1 -10935.926,E2 -10935.926} C_VEL
LIN {X 0,Y 404.114,Z 267.766,A -85,B 0,C 180,E1 -10938.634,E2 -10938.634} C_VEL
LIN {X 0,Y 404.153,Z 267.765,A -85,B 0,C 180,E1 -10941.491,E2 -10941.491} C_VEL
LIN {X 0,Y 404.18,Z 267.731,A -85,B 0,C 180,E1 -10944.983,E2 -10944.983} C_VEL
LIN {X 0,Y 404.144,Z 267.766,A -85,B 0,C 180,E1 -10948.554,E2 -10948.554} C_VEL
LIN {X 0,Y 404.192,Z 267.755,A -85,B 0,C 180,E1 -10952,E2 -10952} C_VEL
LIN {X 0,Y 404.171,Z 267.763,A -85,B 0,C 180,E1 -10955.334,E2 -10955.334} C_VEL
LIN {X 0,Y 404.132,Z 267.763,A -85,B 0,C 180,E1 -10958.58,E2 -10958.58} C_VEL
LIN {X 0,Y 404.203,Z 267.759,A -85,B 0,C 180,E1 -10961.762,E2 -10961.762} C_VEL
LIN {X 0,Y 404.199,Z 267.754,A -85,B 0,C 180,E1 -10964.882,E2 -10964.882} C_VEL
LIN {X 0,Y 404.248,Z 267.75,A -85,B 0,C 180,E1 -10967.958,E2 -10967.958} C_VEL
LIN {X 0,Y 404.426,Z 267.732,A -85,B 0,C 180,E1 -10972.1,E2 -10972.1} C_VEL
LIN {X 0,Y 404.416,Z 267.729,A -85,B 0,C 180,E1 -10974.015,E2 -10974.015} C_VEL
LIN {X 0,Y 404.475,Z 267.725,A -85,B 0,C 180,E1 -10978.009,E2 -10978.009} C_VEL
LIN {X 0,Y 404.603,Z 267.707,A -85,B 0,C 180,E1 -10980,E2 -10980} C_VEL
LIN {X 0,Y 404.416,Z 267.719,A -85,B 0,C 180,E1 -10982.989,E2 -10982.989} C_VEL
LIN {X 0,Y 404.389,Z 267.735,A -85,B 0,C 180,E1 -10986.647,E2 -10986.647} C_VEL
LIN {X 0,Y 404.283,Z 267.738,A -85,B 0,C 180,E1 -10989.001,E2 -10989.001} C_VEL
LIN {X 0,Y 404.249,Z 267.752,A -85,B 0,C 180,E1 -10992.042,E2 -10992.042} C_VEL
LIN {X 0,Y 404.201,Z 267.75,A -85,B 0,C 180,E1 -10995.118,E2 -10995.118} C_VEL
LIN {X 0,Y 404.203,Z 267.758,A -85,B 0,C 180,E1 -10998.238,E2 -10998.238} C_VEL
LIN {X 0,Y 404.132,Z 267.762,A -85,B 0,C 180,E1 -11001.42,E2 -11001.42} C_VEL
LIN {X 0,Y 404.171,Z 267.765,A -85,B 0,C 180,E1 -11004.666,E2 -11004.666} C_VEL
LIN {X 0,Y 404.192,Z 267.759,A -85,B 0,C 180,E1 -11008,E2 -11008} C_VEL
LIN {X 0,Y 404.137,Z 267.751,A -85,B 0,C 180,E1 -11011.559,E2 -11011.559} C_VEL
LIN {X 0,Y 404.181,Z 267.741,A -85,B 0,C 180,E1 -11015.017,E2 -11015.017} C_VEL
LIN {X 0,Y 404.158,Z 267.764,A -85,B 0,C 180,E1 -11018.757,E2 -11018.757} C_VEL
LIN {X 0,Y 404.146,Z 267.74,A -85,B 0,C 180,E1 -11021.605,E2 -11021.605} C_VEL
LIN {X 0,Y 404.143,Z 267.768,A -85,B 0,C 180,E1 -11024.523,E2 -11024.523} C_VEL
LIN {X 0,Y 404.137,Z 267.75,A -85,B 0,C 180,E1 -11027.297,E2 -11027.297} C_VEL
LIN {X 0,Y 404.167,Z 267.764,A -85,B 0,C 180,E1 -11029.956,E2 -11029.956} C_VEL
LIN {X 0,Y 404.135,Z 267.764,A -85,B 0,C 180,E1 -11033.126,E2 -11033.126} C_VEL
LIN {X 0,Y 404.144,Z 267.76,A -85,B 0,C 180,E1 -11036.188,E2 -11036.188} C_VEL
LIN {X 0,Y 404.145,Z 267.77,A -85,B 0,C 180,E1 -11039.716,E2 -11039.716} C_VEL
LIN {X 0,Y 404.201,Z 267.865,A -85,B 0,C 180,E1 -11041.507,E2 -11041.507} C_VEL
LIN {X 0,Y 406.277,Z 277.049,A -85,B 0,C 180,E1 -11043.731,E2 -11043.731} C_VEL
LIN {X 0,Y 408.282,Z 287.597,A -85,B 0,C 180,E1 -11046.094,E2 -11046.094} C_VEL
LIN {X 0,Y 408.759,Z 289.934,A -85,B 0,C 180,E1 -11046.23,E2 -11046.23} C_VEL
LIN {X 0,Y 413.988,Z 315.228,A -85,B 0,C 180,E1 -11047.018,E2 -11047.018} C_VEL
LIN {X 0,Y 412.647,Z 404.621,A -85,B 0,C 180,E1 -11048.586,E2 -11048.586} C_VEL
LIN {X 0,Y 412.148,Z 426.998,A -85,B 0,C 180,E1 -11049.017,E2 -11049.017} C_VEL
LIN {X 0,Y 411.502,Z 441.668,A -85,B 0,C 180,E1 -11049.506,E2 -11049.506} C_VEL
LIN {X 0,Y 410.817,Z 454.702,A -85,B 0,C 180,E1 -11050.135,E2 -11050.135} C_VEL
LIN {X 0,Y 409.885,Z 468.113,A -85,B 0,C 180,E1 -11050.988,E2 -11050.988} C_VEL
LIN {X 0,Y 408.835,Z 480.349,A -85,B 0,C 180,E1 -11051.976,E2 -11051.976} C_VEL
LIN {X 0,Y 407.771,Z 491.556,A -85,B 0,C 180,E1 -11053.092,E2 -11053.092} C_VEL
LIN {X 0,Y 406.667,Z 502.824,A -85,B 0,C 180,E1 -11054.463,E2 -11054.463} C_VEL
LIN {X 0,Y 405.614,Z 513.121,A -85,B 0,C 180,E1 -11056.002,E2 -11056.002} C_VEL
LIN {X 0,Y 404.917,Z 521.238,A -85,B 0,C 180,E1 -11057.47,E2 -11057.47} C_VEL
LIN {X 0,Y 404.084,Z 529.217,A -85,B 0,C 180,E1 -11059.224,E2 -11059.224} C_VEL
LIN {X 0,Y 403.545,Z 535.64,A -85,B 0,C 180,E1 -11060.982,E2 -11060.982} C_VEL
LIN {X 0,Y 403.186,Z 541.334,A -85,B 0,C 180,E1 -11062.992,E2 -11062.992} C_VEL
LIN {X 0,Y 403.008,Z 544.497,A -85,B 0,C 180,E1 -11064.478,E2 -11064.478} C_VEL
LIN {X 0,Y 402.285,Z 545.989,A -85,B 0,C 180,E1 -11065.286,E2 -11065.286} C_VEL
LIN {X 0,Y 399.327,Z 547.817,A -85,B 0,C 180,E1 -11066.612,E2 -11066.612} C_VEL
LIN {X 0,Y 396.86,Z 548.868,A -85,B 0,C 180,E1 -11067.694,E2 -11067.694} C_VEL
LIN {X 0,Y 395.824,Z 549.398,A -85,B 0,C 180,E1 -11068.536,E2 -11068.536} C_VEL
LIN {X 0,Y 395.75,Z 549.527,A -85,B 0,C 180,E1 -11068.822,E2 -11068.822} C_VEL
LIN {X 0,Y 395.759,Z 549.791,A -85,B 0,C 180,E1 -11070,E2 -11070} C_VEL
LIN {X 0,Y 395.761,Z 549.165,A -85,B 0,C 180,E1 -11072.035,E2 -11072.035} C_VEL
LIN {X 0,Y 395.791,Z 547.203,A -85,B 0,C 180,E1 -11074.073,E2 -11074.073} C_VEL
LIN {X 0,Y 395.998,Z 543.857,A -85,B 0,C 180,E1 -11076.113,E2 -11076.113} C_VEL
LIN {X 0,Y 396.25,Z 539.031,A -85,B 0,C 180,E1 -11078.157,E2 -11078.157} C_VEL
LIN {X 0,Y 396.821,Z 532.568,A -85,B 0,C 180,E1 -11080.201,E2 -11080.201} C_VEL
LIN {X 0,Y 397.51,Z 525.372,A -85,B 0,C 180,E1 -11081.99,E2 -11081.99} C_VEL
LIN {X 0,Y 398.257,Z 517.652,A -85,B 0,C 180,E1 -11083.556,E2 -11083.556} C_VEL
LIN {X 0,Y 399.155,Z 508.776,A -85,B 0,C 180,E1 -11085.052,E2 -11085.052} C_VEL
LIN {X 0,Y 400.337,Z 497.807,A -85,B 0,C 180,E1 -11086.575,E2 -11086.575} C_VEL
LIN {X 0,Y 401.503,Z 486.621,A -85,B 0,C 180,E1 -11087.837,E2 -11087.837} C_VEL
LIN {X 0,Y 402.671,Z 474.244,A -85,B 0,C 180,E1 -11088.969,E2 -11088.969} C_VEL
LIN {X 0,Y 403.719,Z 460.867,A -85,B 0,C 180,E1 -11089.941,E2 -11089.941} C_VEL
LIN {X 0,Y 404.634,Z 446.684,A -85,B 0,C 180,E1 -11090.725,E2 -11090.725} C_VEL
LIN {X 0,Y 405.372,Z 432.461,A -85,B 0,C 180,E1 -11091.284,E2 -11091.284} C_VEL
LIN {X 0,Y 405.877,Z 418.837,A -85,B 0,C 180,E1 -11091.622,E2 -11091.622} C_VEL
LIN {X 0,Y 407.478,Z 316.176,A -85,B 0,C 180,E1 -11093.455,E2 -11093.455} C_VEL
LIN {X 0,Y 402.078,Z 290.393,A -85,B 0,C 180,E1 -11094.284,E2 -11094.284} C_VEL
LIN {X 0,Y 401.225,Z 287.601,A -85,B 0,C 180,E1 -11094.462,E2 -11094.462} C_VEL
LIN {X 0,Y 398.465,Z 274.355,A -85,B 0,C 180,E1 -11097.542,E2 -11097.542} C_VEL
LIN {X 0,Y 397.161,Z 268.73,A -85,B 0,C 180,E1 -11098.973,E2 -11098.973} C_VEL
LIN {X 0,Y 397.077,Z 268.646,A -85,B 0,C 180,E1 -11102.071,E2 -11102.071} C_VEL
LIN {X 0,Y 397.118,Z 268.645,A -85,B 0,C 180,E1 -11105.503,E2 -11105.503} C_VEL
LIN {X 0,Y 397.13,Z 268.636,A -85,B 0,C 180,E1 -11108.861,E2 -11108.861} C_VEL
LIN {X 0,Y 397.067,Z 268.63,A -85,B 0,C 180,E1 -11112.266,E2 -11112.266} C_VEL
LIN {X 0,Y 397.085,Z 268.647,A -85,B 0,C 180,E1 -11115.068,E2 -11115.068} C_VEL
LIN {X 0,Y 397.082,Z 268.623,A -85,B 0,C 180,E1 -11118.017,E2 -11118.017} C_VEL
LIN {X 0,Y 397.133,Z 268.638,A -85,B 0,C 180,E1 -11121.137,E2 -11121.137} C_VEL
LIN {X 0,Y 397.115,Z 268.635,A -85,B 0,C 180,E1 -11124.496,E2 -11124.496} C_VEL
LIN {X 0,Y 397.075,Z 268.625,A -85,B 0,C 180,E1 -11127.928,E2 -11127.928} C_VEL
LIN {X 0,Y 397.121,Z 268.644,A -85,B 0,C 180,E1 -11131.456,E2 -11131.456} C_VEL
LIN {X 0,Y 397.146,Z 268.629,A -85,B 0,C 180,E1 -11134.487,E2 -11134.487} C_VEL
LIN {X 0,Y 397.102,Z 268.645,A -85,B 0,C 180,E1 -11137.085,E2 -11137.085} C_VEL
LIN {X 0,Y 397.141,Z 268.632,A -85,B 0,C 180,E1 -11140.352,E2 -11140.352} C_VEL
LIN {X 0,Y 397.159,Z 268.631,A -85,B 0,C 180,E1 -11143.553,E2 -11143.553} C_VEL
LIN {X 0,Y 397.221,Z 268.626,A -85,B 0,C 180,E1 -11146.702,E2 -11146.702} C_VEL
LIN {X 0,Y 397.211,Z 268.625,A -85,B 0,C 180,E1 -11149.809,E2 -11149.809} C_VEL
LIN {X 0,Y 397.348,Z 268.612,A -85,B 0,C 180,E1 -11152.888,E2 -11152.888} C_VEL
LIN {X 0,Y 397.249,Z 268.626,A -85,B 0,C 180,E1 -11154.925,E2 -11154.925} C_VEL
LIN {X 0,Y 397.444,Z 268.586,A -85,B 0,C 180,E1 -11157.973,E2 -11157.973} C_VEL
LIN {X 0,Y 397.574,Z 268.583,A -85,B 0,C 180,E1 -11160,E2 -11160} C_VEL
LIN {X 0,Y 397.374,Z 268.599,A -85,B 0,C 180,E1 -11163.041,E2 -11163.041} C_VEL
LIN {X 0,Y 397.355,Z 268.611,A -85,B 0,C 180,E1 -11167.112,E2 -11167.112} C_VEL
LIN {X 0,Y 397.21,Z 268.62,A -85,B 0,C 180,E1 -11170.191,E2 -11170.191} C_VEL
LIN {X 0,Y 397.219,Z 268.628,A -85,B 0,C 180,E1 -11173.321,E2 -11173.321} C_VEL
LIN {X 0,Y 397.174,Z 268.626,A -85,B 0,C 180,E1 -11177.155,E2 -11177.155} C_VEL
LIN {X 0,Y 397.095,Z 268.64,A -85,B 0,C 180,E1 -11180.73,E2 -11180.73} C_VEL
LIN {X 0,Y 397.126,Z 268.641,A -85,B 0,C 180,E1 -11184.019,E2 -11184.019} C_VEL
LIN {X 0,Y 397.188,Z 268.625,A -85,B 0,C 180,E1 -11187.391,E2 -11187.391} C_VEL
LIN {X 0,Y 397.081,Z 268.644,A -85,B 0,C 180,E1 -11190.882,E2 -11190.882} C_VEL
LIN {X 0,Y 397.12,Z 268.608,A -85,B 0,C 180,E1 -11194.494,E2 -11194.494} C_VEL
LIN {X 0,Y 397.101,Z 268.645,A -85,B 0,C 180,E1 -11198.275,E2 -11198.275} C_VEL
LIN {X 0,Y 397.084,Z 268.64,A -85,B 0,C 180,E1 -11200.909,E2 -11200.909} C_VEL
LIN {X 0,Y 397.098,Z 268.643,A -85,B 0,C 180,E1 -11203.649,E2 -11203.649} C_VEL
LIN {X 0,Y 397.156,Z 268.635,A -85,B 0,C 180,E1 -11206.513,E2 -11206.513} C_VEL
LIN {X 0,Y 397.12,Z 268.632,A -85,B 0,C 180,E1 -11209.551,E2 -11209.551} C_VEL
LIN {X 0,Y 397.095,Z 268.633,A -85,B 0,C 180,E1 -11212.791,E2 -11212.791} C_VEL
LIN {X 0,Y 397.116,Z 268.633,A -85,B 0,C 180,E1 -11216.283,E2 -11216.283} C_VEL
LIN {X 0,Y 397.132,Z 268.677,A -85,B 0,C 180,E1 -11219.815,E2 -11219.815} C_VEL
LIN {X 0,Y 397.558,Z 270.517,A -85,B 0,C 180,E1 -11220.332,E2 -11220.332} C_VEL
LIN {X 0,Y 400.498,Z 283.316,A -85,B 0,C 180,E1 -11223.283,E2 -11223.283} C_VEL
LIN {X 0,Y 401.732,Z 290.669,A -85,B 0,C 180,E1 -11224.898,E2 -11224.898} C_VEL
LIN {X 0,Y 401.424,Z 294.617,A -85,B 0,C 180,E1 -11225.64,E2 -11225.64} C_VEL
LIN {X 0,Y 406.633,Z 320.616,A -85,B 0,C 180,E1 -11226.49,E2 -11226.49} C_VEL
LIN {X 0,Y 407.372,Z 326.209,A -85,B 0,C 180,E1 -11226.641,E2 -11226.641} C_VEL
LIN {X 0,Y 405.772,Z 425.386,A -85,B 0,C 180,E1 -11228.405,E2 -11228.405} C_VEL
LIN {X 0,Y 405.223,Z 440.139,A -85,B 0,C 180,E1 -11228.775,E2 -11228.775} C_VEL
LIN {X 0,Y 404.464,Z 454.202,A -85,B 0,C 180,E1 -11229.333,E2 -11229.333} C_VEL
LIN {X 0,Y 403.525,Z 468.085,A -85,B 0,C 180,E1 -11230.101,E2 -11230.101} C_VEL
LIN {X 0,Y 402.458,Z 480.845,A -85,B 0,C 180,E1 -11231.02,E2 -11231.02} C_VEL
LIN {X 0,Y 401.318,Z 493.348,A -85,B 0,C 180,E1 -11232.154,E2 -11232.154} C_VEL
LIN {X 0,Y 400.129,Z 504.653,A -85,B 0,C 180,E1 -11233.416,E2 -11233.416} C_VEL
LIN {X 0,Y 398.965,Z 515.723,A -85,B 0,C 180,E1 -11234.94,E2 -11234.94} C_VEL
LIN {X 0,Y 398.046,Z 525.035,A -85,B 0,C 180,E1 -11236.505,E2 -11236.505} C_VEL
LIN {X 0,Y 397.242,Z 533.587,A -85,B 0,C 180,E1 -11238.261,E2 -11238.261} C_VEL
LIN {X 0,Y 396.636,Z 539.733,A -85,B 0,C 180,E1 -11239.794,E2 -11239.794} C_VEL
LIN {X 0,Y 396.148,Z 546.261,A -85,B 0,C 180,E1 -11241.841,E2 -11241.841} C_VEL
LIN {X 0,Y 395.909,Z 551.147,A -85,B 0,C 180,E1 -11243.886,E2 -11243.886} C_VEL
LIN {X 0,Y 395.753,Z 554.543,A -85,B 0,C 180,E1 -11245.927,E2 -11245.927} C_VEL
LIN {X 0,Y 395.716,Z 556.551,A -85,B 0,C 180,E1 -11247.965,E2 -11247.965} C_VEL
LIN {X 0,Y 395.758,Z 557.216,A -85,B 0,C 180,E1 -11250,E2 -11250} C_VEL
LIN {X 0,Y 395.717,Z 556.547,A -85,B 0,C 180,E1 -11252.036,E2 -11252.036} C_VEL
LIN {X 0,Y 395.754,Z 554.537,A -85,B 0,C 180,E1 -11254.073,E2 -11254.073} C_VEL
LIN {X 0,Y 395.909,Z 551.135,A -85,B 0,C 180,E1 -11256.114,E2 -11256.114} C_VEL
LIN {X 0,Y 396.149,Z 546.239,A -85,B 0,C 180,E1 -11258.159,E2 -11258.159} C_VEL
LIN {X 0,Y 396.639,Z 539.706,A -85,B 0,C 180,E1 -11260.206,E2 -11260.206} C_VEL
LIN {X 0,Y 397.336,Z 532.436,A -85,B 0,C 180,E1 -11261.995,E2 -11261.995} C_VEL
LIN {X 0,Y 398.116,Z 524.024,A -85,B 0,C 180,E1 -11263.678,E2 -11263.678} C_VEL
LIN {X 0,Y 399.131,Z 513.98,A -85,B 0,C 180,E1 -11265.315,E2 -11265.315} C_VEL
LIN {X 0,Y 400.261,Z 503.518,A -85,B 0,C 180,E1 -11266.709,E2 -11266.709} C_VEL
LIN {X 0,Y 401.324,Z 493.264,A -85,B 0,C 180,E1 -11267.846,E2 -11267.846} C_VEL
LIN {X 0,Y 402.489,Z 480.744,A -85,B 0,C 180,E1 -11268.978,E2 -11268.978} C_VEL
LIN {X 0,Y 403.629,Z 467.244,A -85,B 0,C 180,E1 -11269.941,E2 -11269.941} C_VEL
LIN {X 0,Y 404.478,Z 454.011,A -85,B 0,C 180,E1 -11270.667,E2 -11270.667} C_VEL
LIN {X 0,Y 405.238,Z 439.879,A -85,B 0,C 180,E1 -11271.225,E2 -11271.225} C_VEL
LIN {X 0,Y 405.72,Z 426.474,A -85,B 0,C 180,E1 -11271.565,E2 -11271.565} C_VEL
LIN {X 0,Y 407.294,Z 324.726,A -85,B 0,C 180,E1 -11273.382,E2 -11273.382} C_VEL
LIN {X 0,Y 401.686,Z 296.161,A -85,B 0,C 180,E1 -11274.274,E2 -11274.274} C_VEL
LIN {X 0,Y 401.423,Z 294.493,A -85,B 0,C 180,E1 -11274.362,E2 -11274.362} C_VEL
LIN {X 0,Y 401.646,Z 289.273,A -85,B 0,C 180,E1 -11275.385,E2 -11275.385} C_VEL
LIN {X 0,Y 399.193,Z 277.358,A -85,B 0,C 180,E1 -11278.058,E2 -11278.058} C_VEL
LIN {X 0,Y 397.147,Z 268.774,A -85,B 0,C 180,E1 -11280.115,E2 -11280.115} C_VEL
LIN {X 0,Y 397.116,Z 268.633,A -85,B 0,C 180,E1 -11283.717,E2 -11283.717} C_VEL
LIN {X 0,Y 397.091,Z 268.634,A -85,B 0,C 180,E1 -11287.208,E2 -11287.208} C_VEL
LIN {X 0,Y 397.098,Z 268.634,A -85,B 0,C 180,E1 -11290.445,E2 -11290.445} C_VEL
LIN {X 0,Y 397.1,Z 268.642,A -85,B 0,C 180,E1 -11293.647,E2 -11293.647} C_VEL
LIN {X 0,Y 397.098,Z 268.644,A -85,B 0,C 180,E1 -11296.52,E2 -11296.52} C_VEL
LIN {X 0,Y 397.11,Z 268.644,A -85,B 0,C 180,E1 -11300.422,E2 -11300.422} C_VEL
LIN {X 0,Y 397.104,Z 268.618,A -85,B 0,C 180,E1 -11304.265,E2 -11304.265} C_VEL
LIN {X 0,Y 397.11,Z 268.619,A -85,B 0,C 180,E1 -11306.727,E2 -11306.727} C_VEL
LIN {X 0,Y 397.128,Z 268.642,A -85,B 0,C 180,E1 -11310.296,E2 -11310.296} C_VEL
LIN {X 0,Y 397.189,Z 268.625,A -85,B 0,C 180,E1 -11312.609,E2 -11312.609} C_VEL
LIN {X 0,Y 397.127,Z 268.641,A -85,B 0,C 180,E1 -11315.981,E2 -11315.981} C_VEL
LIN {X 0,Y 397.132,Z 268.639,A -85,B 0,C 180,E1 -11319.704,E2 -11319.704} C_VEL
LIN {X 0,Y 397.175,Z 268.626,A -85,B 0,C 180,E1 -11322.845,E2 -11322.845} C_VEL
LIN {X 0,Y 397.221,Z 268.628,A -85,B 0,C 180,E1 -11326.703,E2 -11326.703} C_VEL
LIN {X 0,Y 397.21,Z 268.62,A -85,B 0,C 180,E1 -11329.809,E2 -11329.809} C_VEL
LIN {X 0,Y 397.356,Z 268.611,A -85,B 0,C 180,E1 -11332.888,E2 -11332.888} C_VEL
LIN {X 0,Y 397.248,Z 268.62,A -85,B 0,C 180,E1 -11334.925,E2 -11334.925} C_VEL
LIN {X 0,Y 397.444,Z 268.601,A -85,B 0,C 180,E1 -11337.973,E2 -11337.973} C_VEL
LIN {X 0,Y 397.573,Z 268.583,A -85,B 0,C 180,E1 -11340,E2 -11340} C_VEL
LIN {X 0,Y 397.375,Z 268.596,A -85,B 0,C 180,E1 -11343.042,E2 -11343.042} C_VEL
LIN {X 0,Y 397.34,Z 268.611,A -85,B 0,C 180,E1 -11346.644,E2 -11346.644} C_VEL
LIN {X 0,Y 397.245,Z 268.615,A -85,B 0,C 180,E1 -11349.162,E2 -11349.162} C_VEL
LIN {X 0,Y 397.212,Z 268.628,A -85,B 0,C 180,E1 -11352.258,E2 -11352.258} C_VEL
LIN {X 0,Y 397.173,Z 268.626,A -85,B 0,C 180,E1 -11355.392,E2 -11355.392} C_VEL
LIN {X 0,Y 397.156,Z 268.637,A -85,B 0,C 180,E1 -11358.574,E2 -11358.574} C_VEL
LIN {X 0,Y 397.09,Z 268.641,A -85,B 0,C 180,E1 -11361.819,E2 -11361.819} C_VEL
LIN {X 0,Y 397.151,Z 268.633,A -85,B 0,C 180,E1 -11365.132,E2 -11365.132} C_VEL
LIN {X 0,Y 397.158,Z 268.635,A -85,B 0,C 180,E1 -11367.777,E2 -11367.777} C_VEL
LIN {X 0,Y 397.079,Z 268.637,A -85,B 0,C 180,E1 -11370.883,E2 -11370.883} C_VEL
LIN {X 0,Y 397.121,Z 268.612,A -85,B 0,C 180,E1 -11374.494,E2 -11374.494} C_VEL
LIN {X 0,Y 397.105,Z 268.645,A -85,B 0,C 180,E1 -11378.275,E2 -11378.275} C_VEL
LIN {X 0,Y 397.108,Z 268.618,A -85,B 0,C 180,E1 -11380.906,E2 -11380.906} C_VEL
LIN {X 0,Y 397.099,Z 268.64,A -85,B 0,C 180,E1 -11383.649,E2 -11383.649} C_VEL
LIN {X 0,Y 397.102,Z 268.634,A -85,B 0,C 180,E1 -11386.521,E2 -11386.521} C_VEL
LIN {X 0,Y 397.112,Z 268.647,A -85,B 0,C 180,E1 -11390.424,E2 -11390.424} C_VEL
LIN {X 0,Y 397.107,Z 268.647,A -85,B 0,C 180,E1 -11394.266,E2 -11394.266} C_VEL
LIN {X 0,Y 397.114,Z 268.641,A -85,B 0,C 180,E1 -11396.728,E2 -11396.728} C_VEL
LIN {X 0,Y 397.124,Z 268.639,A -85,B 0,C 180,E1 -11400.296,E2 -11400.296} C_VEL
LIN {X 0,Y 397.16,Z 268.806,A -85,B 0,C 180,E1 -11401.171,E2 -11401.171} C_VEL
LIN {X 0,Y 399.188,Z 277.56,A -85,B 0,C 180,E1 -11403.325,E2 -11403.325} C_VEL
LIN {X 0,Y 401.276,Z 287.986,A -85,B 0,C 180,E1 -11405.69,E2 -11405.69} C_VEL
LIN {X 0,Y 402.743,Z 293.2,A -85,B 0,C 180,E1 -11405.913,E2 -11405.913} C_VEL
LIN {X 0,Y 407.425,Z 316.087,A -85,B 0,C 180,E1 -11406.64,E2 -11406.64} C_VEL
LIN {X 0,Y 406.052,Z 404.714,A -85,B 0,C 180,E1 -11408.22,E2 -11408.22} C_VEL
LIN {X 0,Y 405.554,Z 427.08,A -85,B 0,C 180,E1 -11408.659,E2 -11408.659} C_VEL
LIN {X 0,Y 404.868,Z 441.746,A -85,B 0,C 180,E1 -11409.155,E2 -11409.155} C_VEL
LIN {X 0,Y 404.108,Z 455.236,A -85,B 0,C 180,E1 -11409.818,E2 -11409.818} C_VEL
LIN {X 0,Y 403.176,Z 468.186,A -85,B 0,C 180,E1 -11410.659,E2 -11410.659} C_VEL
LIN {X 0,Y 402.077,Z 480.421,A -85,B 0,C 180,E1 -11411.662,E2 -11411.662} C_VEL
LIN {X 0,Y 400.861,Z 492.757,A -85,B 0,C 180,E1 -11412.923,E2 -11412.923} C_VEL
LIN {X 0,Y 399.812,Z 502.894,A -85,B 0,C 180,E1 -11414.189,E2 -11414.189} C_VEL
LIN {X 0,Y 398.7,Z 512.955,A -85,B 0,C 180,E1 -11415.713,E2 -11415.713} C_VEL
LIN {X 0,Y 397.973,Z 521.307,A -85,B 0,C 180,E1 -11417.248,E2 -11417.248} C_VEL
LIN {X 0,Y 397.078,Z 529.286,A -85,B 0,C 180,E1 -11419.032,E2 -11419.032} C_VEL
LIN {X 0,Y 396.513,Z 535.708,A -85,B 0,C 180,E1 -11420.821,E2 -11420.821} C_VEL
LIN {X 0,Y 396.101,Z 541.402,A -85,B 0,C 180,E1 -11422.865,E2 -11422.865} C_VEL
LIN {X 0,Y 395.905,Z 545.542,A -85,B 0,C 180,E1 -11424.908,E2 -11424.908} C_VEL
LIN {X 0,Y 395.734,Z 548.251,A -85,B 0,C 180,E1 -11426.946,E2 -11426.946} C_VEL
LIN {X 0,Y 395.75,Z 549.527,A -85,B 0,C 180,E1 -11428.822,E2 -11428.822} C_VEL
LIN {X 0,Y 395.098,Z 549.832,A -85,B 0,C 180,E1 -11429.67,E2 -11429.67} C_VEL
LIN {X 0,Y 392.204,Z 549.786,A -85,B 0,C 180,E1 -11431.051,E2 -11431.051} C_VEL
LIN {X 0,Y 389.754,Z 549.233,A -85,B 0,C 180,E1 -11432.165,E2 -11432.165} C_VEL
LIN {X 0,Y 388.719,Z 548.503,A -85,B 0,C 180,E1 -11433.022,E2 -11433.022} C_VEL
LIN {X 0,Y 388.646,Z 548.197,A -85,B 0,C 180,E1 -11433.311,E2 -11433.311} C_VEL
LIN {X 0,Y 388.83,Z 545.773,A -85,B 0,C 180,E1 -11435.185,E2 -11435.185} C_VEL
LIN {X 0,Y 389.031,Z 541.703,A -85,B 0,C 180,E1 -11437.265,E2 -11437.265} C_VEL
LIN {X 0,Y 389.451,Z 536.08,A -85,B 0,C 180,E1 -11439.347,E2 -11439.347} C_VEL
LIN {X 0,Y 390.015,Z 529.732,A -85,B 0,C 180,E1 -11441.169,E2 -11441.169} C_VEL
LIN {X 0,Y 390.948,Z 521.836,A -85,B 0,C 180,E1 -11442.985,E2 -11442.985} C_VEL
LIN {X 0,Y 391.755,Z 513.579,A -85,B 0,C 180,E1 -11444.546,E2 -11444.546} C_VEL
LIN {X 0,Y 392.862,Z 503.628,A -85,B 0,C 180,E1 -11446.098,E2 -11446.098} C_VEL
LIN {X 0,Y 394.094,Z 492.551,A -85,B 0,C 180,E1 -11447.513,E2 -11447.513} C_VEL
LIN {X 0,Y 395.273,Z 481.522,A -85,B 0,C 180,E1 -11448.665,E2 -11448.665} C_VEL
LIN {X 0,Y 396.493,Z 468.523,A -85,B 0,C 180,E1 -11449.76,E2 -11449.76} C_VEL
LIN {X 0,Y 397.443,Z 455.812,A -85,B 0,C 180,E1 -11450.606,E2 -11450.606} C_VEL
LIN {X 0,Y 398.291,Z 441.801,A -85,B 0,C 180,E1 -11451.308,E2 -11451.308} C_VEL
LIN {X 0,Y 398.986,Z 427.112,A -85,B 0,C 180,E1 -11451.811,E2 -11451.811} C_VEL
LIN {X 0,Y 399.574,Z 402.924,A -85,B 0,C 180,E1 -11452.287,E2 -11452.287} C_VEL
LIN {X 0,Y 400.914,Z 316.913,A -85,B 0,C 180,E1 -11453.849,E2 -11453.849} C_VEL
LIN {X 0,Y 395.753,Z 292.456,A -85,B 0,C 180,E1 -11454.658,E2 -11454.658} C_VEL
LIN {X 0,Y 394.105,Z 288.027,A -85,B 0,C 180,E1 -11454.887,E2 -11454.887} C_VEL
LIN {X 0,Y 391.777,Z 276.806,A -85,B 0,C 180,E1 -11457.511,E2 -11457.511} C_VEL
LIN {X 0,Y 390.11,Z 269.602,A -85,B 0,C 180,E1 -11459.363,E2 -11459.363} C_VEL
LIN {X 0,Y 390.042,Z 269.526,A -85,B 0,C 180,E1 -11462.721,E2 -11462.721} C_VEL
LIN {X 0,Y 390.054,Z 269.528,A -85,B 0,C 180,E1 -11465.825,E2 -11465.825} C_VEL
LIN {X 0,Y 390.068,Z 269.519,A -85,B 0,C 180,E1 -11469.218,E2 -11469.218} C_VEL
LIN {X 0,Y 390.041,Z 269.505,A -85,B 0,C 180,E1 -11472.374,E2 -11472.374} C_VEL
LIN {X 0,Y 390.042,Z 269.528,A -85,B 0,C 180,E1 -11475.354,E2 -11475.354} C_VEL
LIN {X 0,Y 390.046,Z 269.497,A -85,B 0,C 180,E1 -11478.188,E2 -11478.188} C_VEL
LIN {X 0,Y 390.09,Z 269.513,A -85,B 0,C 180,E1 -11480.907,E2 -11480.907} C_VEL
LIN {X 0,Y 390.08,Z 269.504,A -85,B 0,C 180,E1 -11484.792,E2 -11484.792} C_VEL
LIN {X 0,Y 390.021,Z 269.509,A -85,B 0,C 180,E1 -11488.495,E2 -11488.495} C_VEL
LIN {X 0,Y 390.111,Z 269.514,A -85,B 0,C 180,E1 -11492.069,E2 -11492.069} C_VEL
LIN {X 0,Y 390.074,Z 269.52,A -85,B 0,C 180,E1 -11495.519,E2 -11495.519} C_VEL
LIN {X 0,Y 390.048,Z 269.514,A -85,B 0,C 180,E1 -11498.877,E2 -11498.877} C_VEL
LIN {X 0,Y 390.121,Z 269.513,A -85,B 0,C 180,E1 -11502.166,E2 -11502.166} C_VEL
LIN {X 0,Y 390.136,Z 269.502,A -85,B 0,C 180,E1 -11505.392,E2 -11505.392} C_VEL
LIN {X 0,Y 390.142,Z 269.514,A -85,B 0,C 180,E1 -11508.571,E2 -11508.571} C_VEL
LIN {X 0,Y 390.3,Z 269.48,A -85,B 0,C 180,E1 -11512.031,E2 -11512.031} C_VEL
LIN {X 0,Y 390.221,Z 269.502,A -85,B 0,C 180,E1 -11514.833,E2 -11514.833} C_VEL
LIN {X 0,Y 390.412,Z 269.461,A -85,B 0,C 180,E1 -11517.937,E2 -11517.937} C_VEL
LIN {X 0,Y 390.543,Z 269.458,A -85,B 0,C 180,E1 -11520,E2 -11520} C_VEL
LIN {X 0,Y 390.308,Z 269.479,A -85,B 0,C 180,E1 -11523.096,E2 -11523.096} C_VEL
LIN {X 0,Y 390.322,Z 269.486,A -85,B 0,C 180,E1 -11526.202,E2 -11526.202} C_VEL
LIN {X 0,Y 390.306,Z 269.49,A -85,B 0,C 180,E1 -11528.282,E2 -11528.282} C_VEL
LIN {X 0,Y 390.162,Z 269.51,A -85,B 0,C 180,E1 -11532.483,E2 -11532.483} C_VEL
LIN {X 0,Y 390.131,Z 269.507,A -85,B 0,C 180,E1 -11535.677,E2 -11535.677} C_VEL
LIN {X 0,Y 390.098,Z 269.516,A -85,B 0,C 180,E1 -11538.922,E2 -11538.922} C_VEL
LIN {X 0,Y 390.032,Z 269.516,A -85,B 0,C 180,E1 -11542.235,E2 -11542.235} C_VEL
LIN {X 0,Y 390.112,Z 269.517,A -85,B 0,C 180,E1 -11545.744,E2 -11545.744} C_VEL
LIN {X 0,Y 390.059,Z 269.519,A -85,B 0,C 180,E1 -11549.109,E2 -11549.109} C_VEL
LIN {X 0,Y 390.039,Z 269.506,A -85,B 0,C 180,E1 -11552.722,E2 -11552.722} C_VEL
LIN {X 0,Y 390.051,Z 269.498,A -85,B 0,C 180,E1 -11555.826,E2 -11555.826} C_VEL
LIN {X 0,Y 390.067,Z 269.521,A -85,B 0,C 180,E1 -11559.219,E2 -11559.219} C_VEL
LIN {X 0,Y 390.038,Z 269.524,A -85,B 0,C 180,E1 -11562.375,E2 -11562.375} C_VEL
LIN {X 0,Y 390.098,Z 269.516,A -85,B 0,C 180,E1 -11566.107,E2 -11566.107} C_VEL
LIN {X 0,Y 390.079,Z 269.504,A -85,B 0,C 180,E1 -11569.175,E2 -11569.175} C_VEL
LIN {X 0,Y 390.044,Z 269.512,A -85,B 0,C 180,E1 -11572.449,E2 -11572.449} C_VEL
LIN {X 0,Y 390.065,Z 269.512,A -85,B 0,C 180,E1 -11576.046,E2 -11576.046} C_VEL
LIN {X 0,Y 390.073,Z 269.654,A -85,B 0,C 180,E1 -11579.48,E2 -11579.48} C_VEL
LIN {X 0,Y 393.119,Z 282.426,A -85,B 0,C 180,E1 -11582.564,E2 -11582.564} C_VEL
LIN {X 0,Y 394.861,Z 291.942,A -85,B 0,C 180,E1 -11584.713,E2 -11584.713} C_VEL
LIN {X 0,Y 394.681,Z 294.476,A -85,B 0,C 180,E1 -11585.189,E2 -11585.189} C_VEL
LIN {X 0,Y 399.417,Z 317.917,A -85,B 0,C 180,E1 -11585.988,E2 -11585.988} C_VEL
LIN {X 0,Y 400.863,Z 327.208,A -85,B 0,C 180,E1 -11586.258,E2 -11586.258} C_VEL
LIN {X 0,Y 399.059,Z 428.347,A -85,B 0,C 180,E1 -11588.091,E2 -11588.091} C_VEL
LIN {X 0,Y 398.471,Z 442.83,A -85,B 0,C 180,E1 -11588.499,E2 -11588.499} C_VEL
LIN {X 0,Y 397.656,Z 456.745,A -85,B 0,C 180,E1 -11589.098,E2 -11589.098} C_VEL
LIN {X 0,Y 396.685,Z 470.082,A -85,B 0,C 180,E1 -11589.883,E2 -11589.883} C_VEL
LIN {X 0,Y 395.617,Z 482.36,A -85,B 0,C 180,E1 -11590.814,E2 -11590.814} C_VEL
LIN {X 0,Y 394.398,Z 494.523,A -85,B 0,C 180,E1 -11591.964,E2 -11591.964} C_VEL
LIN {X 0,Y 393.292,Z 504.589,A -85,B 0,C 180,E1 -11593.12,E2 -11593.12} C_VEL
LIN {X 0,Y 392.069,Z 515.659,A -85,B 0,C 180,E1 -11594.669,E2 -11594.669} C_VEL
LIN {X 0,Y 391.179,Z 524.362,A -85,B 0,C 180,E1 -11596.145,E2 -11596.145} C_VEL
LIN {X 0,Y 390.355,Z 532.403,A -85,B 0,C 180,E1 -11597.787,E2 -11597.787} C_VEL
LIN {X 0,Y 389.59,Z 539.667,A -85,B 0,C 180,E1 -11599.608,E2 -11599.608} C_VEL
LIN {X 0,Y 389.091,Z 546.195,A -85,B 0,C 180,E1 -11601.692,E2 -11601.692} C_VEL
LIN {X 0,Y 388.833,Z 551.081,A -85,B 0,C 180,E1 -11603.774,E2 -11603.774} C_VEL
LIN {X 0,Y 388.679,Z 554.477,A -85,B 0,C 180,E1 -11605.853,E2 -11605.853} C_VEL
LIN {X 0,Y 388.613,Z 556.484,A -85,B 0,C 180,E1 -11607.927,E2 -11607.927} C_VEL
LIN {X 0,Y 388.671,Z 557.149,A -85,B 0,C 180,E1 -11610,E2 -11610} C_VEL
LIN {X 0,Y 388.614,Z 556.48,A -85,B 0,C 180,E1 -11612.073,E2 -11612.073} C_VEL
LIN {X 0,Y 388.68,Z 554.47,A -85,B 0,C 180,E1 -11614.148,E2 -11614.148} C_VEL
LIN {X 0,Y 388.833,Z 551.067,A -85,B 0,C 180,E1 -11616.226,E2 -11616.226} C_VEL
LIN {X 0,Y 389.092,Z 546.171,A -85,B 0,C 180,E1 -11618.308,E2 -11618.308} C_VEL
LIN {X 0,Y 389.592,Z 539.637,A -85,B 0,C 180,E1 -11620.393,E2 -11620.393} C_VEL
LIN {X 0,Y 390.359,Z 532.368,A -85,B 0,C 180,E1 -11622.213,E2 -11622.213} C_VEL
LIN {X 0,Y 391.118,Z 524.514,A -85,B 0,C 180,E1 -11623.819,E2 -11623.819} C_VEL
LIN {X 0,Y 392.074,Z 515.604,A -85,B 0,C 180,E1 -11625.331,E2 -11625.331} C_VEL
LIN {X 0,Y 393.055,Z 506.489,A -85,B 0,C 180,E1 -11626.624,E2 -11626.624} C_VEL
LIN {X 0,Y 394.255,Z 495.615,A -85,B 0,C 180,E1 -11627.908,E2 -11627.908} C_VEL
LIN {X 0,Y 395.492,Z 483.711,A -85,B 0,C 180,E1 -11629.058,E2 -11629.058} C_VEL
LIN {X 0,Y 396.671,Z 470.611,A -85,B 0,C 180,E1 -11630.07,E2 -11630.07} C_VEL
LIN {X 0,Y 397.593,Z 457.825,A -85,B 0,C 180,E1 -11630.838,E2 -11630.838} C_VEL
LIN {X 0,Y 398.452,Z 444.378,A -85,B 0,C 180,E1 -11631.434,E2 -11631.434} C_VEL
LIN {X 0,Y 398.963,Z 430.904,A -85,B 0,C 180,E1 -11631.847,E2 -11631.847} C_VEL
LIN {X 0,Y 400.824,Z 326.602,A -85,B 0,C 180,E1 -11633.745,E2 -11633.745} C_VEL
LIN {X 0,Y 398.48,Z 313.63,A -85,B 0,C 180,E1 -11634.144,E2 -11634.144} C_VEL
LIN {X 0,Y 394.712,Z 294.482,A -85,B 0,C 180,E1 -11634.796,E2 -11634.796} C_VEL
LIN {X 0,Y 394.715,Z 290.543,A -85,B 0,C 180,E1 -11635.58,E2 -11635.58} C_VEL
LIN {X 0,Y 392.213,Z 278.559,A -85,B 0,C 180,E1 -11638.327,E2 -11638.327} C_VEL
LIN {X 0,Y 390.074,Z 269.627,A -85,B 0,C 180,E1 -11640.521,E2 -11640.521} C_VEL
LIN {X 0,Y 390.066,Z 269.512,A -85,B 0,C 180,E1 -11644.024,E2 -11644.024} C_VEL
LIN {X 0,Y 390.04,Z 269.513,A -85,B 0,C 180,E1 -11647.55,E2 -11647.55} C_VEL
LIN {X 0,Y 390.053,Z 269.507,A -85,B 0,C 180,E1 -11650.821,E2 -11650.821} C_VEL
LIN {X 0,Y 390.053,Z 269.522,A -85,B 0,C 180,E1 -11653.886,E2 -11653.886} C_VEL
LIN {X 0,Y 390.053,Z 269.524,A -85,B 0,C 180,E1 -11656.789,E2 -11656.789} C_VEL
LIN {X 0,Y 390.052,Z 269.515,A -85,B 0,C 180,E1 -11659.56,E2 -11659.56} C_VEL
LIN {X 0,Y 390.041,Z 269.52,A -85,B 0,C 180,E1 -11662.448,E2 -11662.448} C_VEL
LIN {X 0,Y 390.063,Z 269.487,A -85,B 0,C 180,E1 -11666.045,E2 -11666.045} C_VEL
LIN {X 0,Y 390.047,Z 269.525,A -85,B 0,C 180,E1 -11669.867,E2 -11669.867} C_VEL
LIN {X 0,Y 390.107,Z 269.507,A -85,B 0,C 180,E1 -11673.231,E2 -11673.231} C_VEL
LIN {X 0,Y 390.1,Z 269.509,A -85,B 0,C 180,E1 -11676.75,E2 -11676.75} C_VEL
LIN {X 0,Y 390.097,Z 269.519,A -85,B 0,C 180,E1 -11679.983,E2 -11679.983} C_VEL
LIN {X 0,Y 390.131,Z 269.502,A -85,B 0,C 180,E1 -11683.248,E2 -11683.248} C_VEL
LIN {X 0,Y 390.187,Z 269.504,A -85,B 0,C 180,E1 -11686.561,E2 -11686.561} C_VEL
LIN {X 0,Y 390.197,Z 269.496,A -85,B 0,C 180,E1 -11690.671,E2 -11690.671} C_VEL
LIN {X 0,Y 390.311,Z 269.488,A -85,B 0,C 180,E1 -11692.759,E2 -11692.759} C_VEL
LIN {X 0,Y 390.22,Z 269.495,A -85,B 0,C 180,E1 -11694.833,E2 -11694.833} C_VEL
LIN {X 0,Y 390.413,Z 269.478,A -85,B 0,C 180,E1 -11697.937,E2 -11697.937} C_VEL
LIN {X 0,Y 390.542,Z 269.459,A -85,B 0,C 180,E1 -11700,E2 -11700} C_VEL
LIN {X 0,Y 390.309,Z 269.476,A -85,B 0,C 180,E1 -11703.097,E2 -11703.097} C_VEL
LIN {X 0,Y 390.295,Z 269.488,A -85,B 0,C 180,E1 -11706.64,E2 -11706.64} C_VEL
LIN {X 0,Y 390.198,Z 269.493,A -85,B 0,C 180,E1 -11709.329,E2 -11709.329} C_VEL
LIN {X 0,Y 390.164,Z 269.507,A -85,B 0,C 180,E1 -11712.483,E2 -11712.483} C_VEL
LIN {X 0,Y 390.133,Z 269.504,A -85,B 0,C 180,E1 -11715.677,E2 -11715.677} C_VEL
LIN {X 0,Y 390.099,Z 269.519,A -85,B 0,C 180,E1 -11718.923,E2 -11718.923} C_VEL
LIN {X 0,Y 390.033,Z 269.52,A -85,B 0,C 180,E1 -11722.235,E2 -11722.235} C_VEL
LIN {X 0,Y 390.113,Z 269.504,A -85,B 0,C 180,E1 -11725.744,E2 -11725.744} C_VEL
LIN {X 0,Y 390.06,Z 269.523,A -85,B 0,C 180,E1 -11729.11,E2 -11729.11} C_VEL
LIN {X 0,Y 390.039,Z 269.491,A -85,B 0,C 180,E1 -11732.722,E2 -11732.722} C_VEL
LIN {X 0,Y 390.053,Z 269.514,A -85,B 0,C 180,E1 -11735.826,E2 -11735.826} C_VEL
LIN {X 0,Y 390.07,Z 269.513,A -85,B 0,C 180,E1 -11739.22,E2 -11739.22} C_VEL
LIN {X 0,Y 390.052,Z 269.499,A -85,B 0,C 180,E1 -11742.377,E2 -11742.377} C_VEL
LIN {X 0,Y 390.054,Z 269.52,A -85,B 0,C 180,E1 -11746.114,E2 -11746.114} C_VEL
LIN {X 0,Y 390.055,Z 269.521,A -85,B 0,C 180,E1 -11749.561,E2 -11749.561} C_VEL
LIN {X 0,Y 390.042,Z 269.513,A -85,B 0,C 180,E1 -11752.45,E2 -11752.45} C_VEL
LIN {X 0,Y 390.067,Z 269.513,A -85,B 0,C 180,E1 -11755.976,E2 -11755.976} C_VEL
LIN {X 0,Y 390.046,Z 269.527,A -85,B 0,C 180,E1 -11759.87,E2 -11759.87} C_VEL
LIN {X 0,Y 390.12,Z 269.606,A -85,B 0,C 180,E1 -11760.748,E2 -11760.748} C_VEL
LIN {X 0,Y 392.266,Z 278.906,A -85,B 0,C 180,E1 -11763.104,E2 -11763.104} C_VEL
LIN {X 0,Y 394.065,Z 287.913,A -85,B 0,C 180,E1 -11765.199,E2 -11765.199} C_VEL
LIN {X 0,Y 396.103,Z 293.636,A -85,B 0,C 180,E1 -11765.49,E2 -11765.49} C_VEL
LIN {X 0,Y 400.978,Z 317.526,A -85,B 0,C 180,E1 -11766.267,E2 -11766.267} C_VEL
LIN {X 0,Y 399.095,Z 423.468,A -85,B 0,C 180,E1 -11768.195,E2 -11768.195} C_VEL
LIN {X 0,Y 398.485,Z 438,A -85,B 0,C 180,E1 -11768.635,E2 -11768.635} C_VEL
LIN {X 0,Y 397.721,Z 451.251,A -85,B 0,C 180,E1 -11769.237,E2 -11769.237} C_VEL
LIN {X 0,Y 396.814,Z 464.257,A -85,B 0,C 180,E1 -11770.03,E2 -11770.03} C_VEL
LIN {X 0,Y 395.805,Z 476.221,A -85,B 0,C 180,E1 -11770.958,E2 -11770.958} C_VEL
LIN {X 0,Y 394.57,Z 488.183,A -85,B 0,C 180,E1 -11772.107,E2 -11772.107} C_VEL
LIN {X 0,Y 393.395,Z 499.094,A -85,B 0,C 180,E1 -11773.391,E2 -11773.391} C_VEL
LIN {X 0,Y 392.13,Z 509.859,A -85,B 0,C 180,E1 -11774.937,E2 -11774.937} C_VEL
LIN {X 0,Y 391.257,Z 518.741,A -85,B 0,C 180,E1 -11776.496,E2 -11776.496} C_VEL
LIN {X 0,Y 390.294,Z 527.247,A -85,B 0,C 180,E1 -11778.312,E2 -11778.312} C_VEL
LIN {X 0,Y 389.637,Z 534.098,A -85,B 0,C 180,E1 -11780.134,E2 -11780.134} C_VEL
LIN {X 0,Y 389.21,Z 538.827,A -85,B 0,C 180,E1 -11781.694,E2 -11781.694} C_VEL
LIN {X 0,Y 388.923,Z 543.725,A -85,B 0,C 180,E1 -11783.776,E2 -11783.776} C_VEL
LIN {X 0,Y 388.718,Z 547.136,A -85,B 0,C 180,E1 -11785.853,E2 -11785.853} C_VEL
LIN {X 0,Y 388.66,Z 549.162,A -85,B 0,C 180,E1 -11787.927,E2 -11787.927} C_VEL
LIN {X 0,Y 388.672,Z 549.858,A -85,B 0,C 180,E1 -11790,E2 -11790} C_VEL
LIN {X 0,Y 388.659,Z 549.232,A -85,B 0,C 180,E1 -11792.072,E2 -11792.072} C_VEL
LIN {X 0,Y 388.646,Z 548.197,A -85,B 0,C 180,E1 -11793.311,E2 -11793.311} C_VEL
LIN {X 0,Y 388.02,Z 547.262,A -85,B 0,C 180,E1 -11794.164,E2 -11794.164} C_VEL
LIN {X 0,Y 385.257,Z 545.276,A -85,B 0,C 180,E1 -11795.546,E2 -11795.546} C_VEL
LIN {X 0,Y 382.961,Z 543.322,A -85,B 0,C 180,E1 -11796.649,E2 -11796.649} C_VEL
LIN {X 0,Y 382.052,Z 541.565,A -85,B 0,C 180,E1 -11797.489,E2 -11797.489} C_VEL
LIN {X 0,Y 382.02,Z 540.904,A -85,B 0,C 180,E1 -11797.77,E2 -11797.77} C_VEL
LIN {X 0,Y 382.423,Z 536.146,A -85,B 0,C 180,E1 -11799.52,E2 -11799.52} C_VEL
LIN {X 0,Y 383.026,Z 529.797,A -85,B 0,C 180,E1 -11801.376,E2 -11801.376} C_VEL
LIN {X 0,Y 384.003,Z 521.901,A -85,B 0,C 180,E1 -11803.225,E2 -11803.225} C_VEL
LIN {X 0,Y 384.858,Z 513.643,A -85,B 0,C 180,E1 -11804.812,E2 -11804.812} C_VEL
LIN {X 0,Y 386.031,Z 503.691,A -85,B 0,C 180,E1 -11806.39,E2 -11806.39} C_VEL
LIN {X 0,Y 387.312,Z 492.614,A -85,B 0,C 180,E1 -11807.83,E2 -11807.83} C_VEL
LIN {X 0,Y 388.548,Z 481.584,A -85,B 0,C 180,E1 -11809,E2 -11809} C_VEL
LIN {X 0,Y 389.72,Z 469.611,A -85,B 0,C 180,E1 -11810.037,E2 -11810.037} C_VEL
LIN {X 0,Y 390.808,Z 455.837,A -85,B 0,C 180,E1 -11810.974,E2 -11810.974} C_VEL
LIN {X 0,Y 391.683,Z 441.856,A -85,B 0,C 180,E1 -11811.685,E2 -11811.685} C_VEL
LIN {X 0,Y 392.42,Z 427.162,A -85,B 0,C 180,E1 -11812.195,E2 -11812.195} C_VEL
LIN {X 0,Y 393.032,Z 402.965,A -85,B 0,C 180,E1 -11812.678,E2 -11812.678} C_VEL
LIN {X 0,Y 394.421,Z 317.943,A -85,B 0,C 180,E1 -11814.247,E2 -11814.247} C_VEL
LIN {X 0,Y 389.584,Z 294.904,A -85,B 0,C 180,E1 -11815.027,E2 -11815.027} C_VEL
LIN {X 0,Y 386.919,Z 288.057,A -85,B 0,C 180,E1 -11815.385,E2 -11815.385} C_VEL
LIN {X 0,Y 384.587,Z 276.871,A -85,B 0,C 180,E1 -11818.07,E2 -11818.07} C_VEL
LIN {X 0,Y 383.051,Z 270.501,A -85,B 0,C 180,E1 -11819.753,E2 -11819.753} C_VEL
LIN {X 0,Y 383.002,Z 270.398,A -85,B 0,C 180,E1 -11823.4,E2 -11823.4} C_VEL
LIN {X 0,Y 383.03,Z 270.4,A -85,B 0,C 180,E1 -11826.164,E2 -11826.164} C_VEL
LIN {X 0,Y 383.007,Z 270.403,A -85,B 0,C 180,E1 -11829.957,E2 -11829.957} C_VEL
LIN {X 0,Y 383.002,Z 270.381,A -85,B 0,C 180,E1 -11832.778,E2 -11832.778} C_VEL
LIN {X 0,Y 382.995,Z 270.4,A -85,B 0,C 180,E1 -11835.789,E2 -11835.789} C_VEL
LIN {X 0,Y 383.003,Z 270.372,A -85,B 0,C 180,E1 -11838.792,E2 -11838.792} C_VEL
LIN {X 0,Y 382.999,Z 270.403,A -85,B 0,C 180,E1 -11842.095,E2 -11842.095} C_VEL
LIN {X 0,Y 383.013,Z 270.374,A -85,B 0,C 180,E1 -11845.331,E2 -11845.331} C_VEL
LIN {X 0,Y 382.98,Z 270.391,A -85,B 0,C 180,E1 -11849.081,E2 -11849.081} C_VEL
LIN {X 0,Y 383.05,Z 270.394,A -85,B 0,C 180,E1 -11852.697,E2 -11852.697} C_VEL
LIN {X 0,Y 383.046,Z 270.391,A -85,B 0,C 180,E1 -11855.039,E2 -11855.039} C_VEL
LIN {X 0,Y 382.986,Z 270.397,A -85,B 0,C 180,E1 -11858.468,E2 -11858.468} C_VEL
LIN {X 0,Y 383.055,Z 270.393,A -85,B 0,C 180,E1 -11861.826,E2 -11861.826} C_VEL
LIN {X 0,Y 383.102,Z 270.376,A -85,B 0,C 180,E1 -11865.118,E2 -11865.118} C_VEL
LIN {X 0,Y 383.091,Z 270.39,A -85,B 0,C 180,E1 -11868.358,E2 -11868.358} C_VEL
LIN {X 0,Y 383.257,Z 270.357,A -85,B 0,C 180,E1 -11871.974,E2 -11871.974} C_VEL
LIN {X 0,Y 383.192,Z 270.379,A -85,B 0,C 180,E1 -11874.738,E2 -11874.738} C_VEL
LIN {X 0,Y 383.38,Z 270.336,A -85,B 0,C 180,E1 -11877.899,E2 -11877.899} C_VEL
LIN {X 0,Y 383.513,Z 270.334,A -85,B 0,C 180,E1 -11880,E2 -11880} C_VEL
LIN {X 0,Y 383.244,Z 270.358,A -85,B 0,C 180,E1 -11883.154,E2 -11883.154} C_VEL
LIN {X 0,Y 383.279,Z 270.365,A -85,B 0,C 180,E1 -11886.316,E2 -11886.316} C_VEL
LIN {X 0,Y 383.252,Z 270.366,A -85,B 0,C 180,E1 -11888.436,E2 -11888.436} C_VEL
LIN {X 0,Y 383.089,Z 270.382,A -85,B 0,C 180,E1 -11891.642,E2 -11891.642} C_VEL
LIN {X 0,Y 383.102,Z 270.383,A -85,B 0,C 180,E1 -11894.882,E2 -11894.882} C_VEL
LIN {X 0,Y 383.081,Z 270.388,A -85,B 0,C 180,E1 -11898.173,E2 -11898.173} C_VEL
LIN {X 0,Y 382.985,Z 270.396,A -85,B 0,C 180,E1 -11901.531,E2 -11901.531} C_VEL
LIN {X 0,Y 383.045,Z 270.394,A -85,B 0,C 180,E1 -11904.961,E2 -11904.961} C_VEL
LIN {X 0,Y 383.043,Z 270.394,A -85,B 0,C 180,E1 -11908.492,E2 -11908.492} C_VEL
LIN {X 0,Y 383.007,Z 270.386,A -85,B 0,C 180,E1 -11912.15,E2 -11912.15} C_VEL
LIN {X 0,Y 383.012,Z 270.363,A -85,B 0,C 180,E1 -11914.669,E2 -11914.669} C_VEL
LIN {X 0,Y 382.996,Z 270.402,A -85,B 0,C 180,E1 -11917.905,E2 -11917.905} C_VEL
LIN {X 0,Y 382.979,Z 270.399,A -85,B 0,C 180,E1 -11921.348,E2 -11921.348} C_VEL
LIN {X 0,Y 383.002,Z 270.398,A -85,B 0,C 180,E1 -11924.306,E2 -11924.306} C_VEL
LIN {X 0,Y 383.071,Z 270.381,A -85,B 0,C 180,E1 -11927.25,E2 -11927.25} C_VEL
LIN {X 0,Y 383.019,Z 270.399,A -85,B 0,C 180,E1 -11930.413,E2 -11930.413} C_VEL
LIN {X 0,Y 383.024,Z 270.394,A -85,B 0,C 180,E1 -11934.045,E2 -11934.045} C_VEL
LIN {X 0,Y 382.985,Z 270.404,A -85,B 0,C 180,E1 -11937.579,E2 -11937.579} C_VEL
LIN {X 0,Y 383.028,Z 270.552,A -85,B 0,C 180,E1 -11939.086,E2 -11939.086} C_VEL
LIN {X 0,Y 386.196,Z 283.829,A -85,B 0,C 180,E1 -11942.353,E2 -11942.353} C_VEL
LIN {X 0,Y 387.967,Z 293.202,A -85,B 0,C 180,E1 -11944.516,E2 -11944.516} C_VEL
LIN {X 0,Y 388.004,Z 294.843,A -85,B 0,C 180,E1 -11944.76,E2 -11944.76} C_VEL
LIN {X 0,Y 393.465,Z 321.871,A -85,B 0,C 180,E1 -11945.68,E2 -11945.68} C_VEL
LIN {X 0,Y 394.364,Z 327.318,A -85,B 0,C 180,E1 -11945.845,E2 -11945.845} C_VEL
LIN {X 0,Y 392.448,Z 429.802,A -85,B 0,C 180,E1 -11947.737,E2 -11947.737} C_VEL
LIN {X 0,Y 391.84,Z 443.689,A -85,B 0,C 180,E1 -11948.151,E2 -11948.151} C_VEL
LIN {X 0,Y 390.962,Z 457.955,A -85,B 0,C 180,E1 -11948.792,E2 -11948.792} C_VEL
LIN {X 0,Y 389.878,Z 471.597,A -85,B 0,C 180,E1 -11949.635,E2 -11949.635} C_VEL
LIN {X 0,Y 388.767,Z 483.747,A -85,B 0,C 180,E1 -11950.6,E2 -11950.6} C_VEL
LIN {X 0,Y 387.489,Z 495.635,A -85,B 0,C 180,E1 -11951.768,E2 -11951.768} C_VEL
LIN {X 0,Y 386.243,Z 506.493,A -85,B 0,C 180,E1 -11953.075,E2 -11953.075} C_VEL
LIN {X 0,Y 384.994,Z 517.223,A -85,B 0,C 180,E1 -11954.652,E2 -11954.652} C_VEL
LIN {X 0,Y 384.04,Z 526.083,A -85,B 0,C 180,E1 -11956.238,E2 -11956.238} C_VEL
LIN {X 0,Y 383.15,Z 534.574,A -85,B 0,C 180,E1 -11958.091,E2 -11958.091} C_VEL
LIN {X 0,Y 382.403,Z 541.414,A -85,B 0,C 180,E1 -11959.945,E2 -11959.945} C_VEL
LIN {X 0,Y 382.025,Z 546.129,A -85,B 0,C 180,E1 -11961.537,E2 -11961.537} C_VEL
LIN {X 0,Y 381.764,Z 551.015,A -85,B 0,C 180,E1 -11963.659,E2 -11963.659} C_VEL
LIN {X 0,Y 381.606,Z 554.41,A -85,B 0,C 180,E1 -11965.775,E2 -11965.775} C_VEL
LIN {X 0,Y 381.511,Z 556.418,A -85,B 0,C 180,E1 -11967.889,E2 -11967.889} C_VEL
LIN {X 0,Y 381.571,Z 557.082,A -85,B 0,C 180,E1 -11970,E2 -11970} C_VEL
LIN {X 0,Y 381.511,Z 556.413,A -85,B 0,C 180,E1 -11972.111,E2 -11972.111} C_VEL
LIN {X 0,Y 381.607,Z 554.403,A -85,B 0,C 180,E1 -11974.225,E2 -11974.225} C_VEL
LIN {X 0,Y 381.764,Z 551,A -85,B 0,C 180,E1 -11976.342,E2 -11976.342} C_VEL
LIN {X 0,Y 382.026,Z 546.103,A -85,B 0,C 180,E1 -11978.463,E2 -11978.463} C_VEL
LIN {X 0,Y 382.418,Z 541.382,A -85,B 0,C 180,E1 -11980.055,E2 -11980.055} C_VEL
LIN {X 0,Y 383.149,Z 534.535,A -85,B 0,C 180,E1 -11981.909,E2 -11981.909} C_VEL
LIN {X 0,Y 383.853,Z 527.39,A -85,B 0,C 180,E1 -11983.499,E2 -11983.499} C_VEL
LIN {X 0,Y 384.8,Z 518.793,A -85,B 0,C 180,E1 -11985.085,E2 -11985.085} C_VEL
LIN {X 0,Y 385.988,Z 508.373,A -85,B 0,C 180,E1 -11986.665,E2 -11986.665} C_VEL
LIN {X 0,Y 387.339,Z 496.72,A -85,B 0,C 180,E1 -11988.102,E2 -11988.102} C_VEL
LIN {X 0,Y 388.627,Z 485.067,A -85,B 0,C 180,E1 -11989.271,E2 -11989.271} C_VEL
LIN {X 0,Y 389.826,Z 472.244,A -85,B 0,C 180,E1 -11990.306,E2 -11990.306} C_VEL
LIN {X 0,Y 390.883,Z 458.904,A -85,B 0,C 180,E1 -11991.144,E2 -11991.144} C_VEL
LIN {X 0,Y 391.787,Z 445.146,A -85,B 0,C 180,E1 -11991.783,E2 -11991.783} C_VEL
LIN {X 0,Y 392.398,Z 430.821,A -85,B 0,C 180,E1 -11992.231,E2 -11992.231} C_VEL
LIN {X 0,Y 394.308,Z 328.784,A -85,B 0,C 180,E1 -11994.118,E2 -11994.118} C_VEL
LIN {X 0,Y 393.947,Z 324.548,A -85,B 0,C 180,E1 -11994.224,E2 -11994.224} C_VEL
LIN {X 0,Y 388.026,Z 294.805,A -85,B 0,C 180,E1 -11995.225,E2 -11995.225} C_VEL
LIN {X 0,Y 387.971,Z 293.167,A -85,B 0,C 180,E1 -11995.479,E2 -11995.479} C_VEL
LIN {X 0,Y 385.867,Z 282.415,A -85,B 0,C 180,E1 -11997.968,E2 -11997.968} C_VEL
LIN {X 0,Y 383.028,Z 270.526,A -85,B 0,C 180,E1 -12000.914,E2 -12000.914} C_VEL
LIN {X 0,Y 383.016,Z 270.397,A -85,B 0,C 180,E1 -12004.667,E2 -12004.667} C_VEL
LIN {X 0,Y 382.996,Z 270.393,A -85,B 0,C 180,E1 -12007.903,E2 -12007.903} C_VEL
LIN {X 0,Y 382.981,Z 270.383,A -85,B 0,C 180,E1 -12011.347,E2 -12011.347} C_VEL
LIN {X 0,Y 382.995,Z 270.405,A -85,B 0,C 180,E1 -12014.303,E2 -12014.303} C_VEL
LIN {X 0,Y 383.006,Z 270.4,A -85,B 0,C 180,E1 -12017.24,E2 -12017.24} C_VEL
LIN {X 0,Y 383.012,Z 270.399,A -85,B 0,C 180,E1 -12020.413,E2 -12020.413} C_VEL
LIN {X 0,Y 383.021,Z 270.373,A -85,B 0,C 180,E1 -12024.044,E2 -12024.044} C_VEL
LIN {X 0,Y 382.985,Z 270.387,A -85,B 0,C 180,E1 -12027.577,E2 -12027.577} C_VEL
LIN {X 0,Y 382.993,Z 270.403,A -85,B 0,C 180,E1 -12030.3,E2 -12030.3} C_VEL
LIN {X 0,Y 383.051,Z 270.385,A -85,B 0,C 180,E1 -12032.698,E2 -12032.698} C_VEL
LIN {X 0,Y 383.027,Z 270.394,A -85,B 0,C 180,E1 -12036.192,E2 -12036.192} C_VEL
LIN {X 0,Y 383.048,Z 270.392,A -85,B 0,C 180,E1 -12039.598,E2 -12039.598} C_VEL
LIN {X 0,Y 383.098,Z 270.379,A -85,B 0,C 180,E1 -12042.931,E2 -12042.931} C_VEL
LIN {X 0,Y 383.118,Z 270.385,A -85,B 0,C 180,E1 -12046.464,E2 -12046.464} C_VEL
LIN {X 0,Y 383.144,Z 270.374,A -85,B 0,C 180,E1 -12050.498,E2 -12050.498} C_VEL
LIN {X 0,Y 383.265,Z 270.366,A -85,B 0,C 180,E1 -12052.625,E2 -12052.625} C_VEL
LIN {X 0,Y 383.192,Z 270.37,A -85,B 0,C 180,E1 -12054.738,E2 -12054.738} C_VEL
LIN {X 0,Y 383.38,Z 270.354,A -85,B 0,C 180,E1 -12057.899,E2 -12057.899} C_VEL
LIN {X 0,Y 383.512,Z 270.335,A -85,B 0,C 180,E1 -12060,E2 -12060} C_VEL
LIN {X 0,Y 383.245,Z 270.356,A -85,B 0,C 180,E1 -12063.154,E2 -12063.154} C_VEL
LIN {X 0,Y 383.255,Z 270.364,A -85,B 0,C 180,E1 -12066.632,E2 -12066.632} C_VEL
LIN {X 0,Y 383.144,Z 270.372,A -85,B 0,C 180,E1 -12069.502,E2 -12069.502} C_VEL
LIN {X 0,Y 383.119,Z 270.38,A -85,B 0,C 180,E1 -12073.536,E2 -12073.536} C_VEL
LIN {X 0,Y 383.088,Z 270.392,A -85,B 0,C 180,E1 -12077.455,E2 -12077.455} C_VEL
LIN {X 0,Y 383.022,Z 270.388,A -85,B 0,C 180,E1 -12080.647,E2 -12080.647} C_VEL
LIN {X 0,Y 383.028,Z 270.397,A -85,B 0,C 180,E1 -12083.808,E2 -12083.808} C_VEL
LIN {X 0,Y 383.074,Z 270.381,A -85,B 0,C 180,E1 -12086.124,E2 -12086.124} C_VEL
LIN {X 0,Y 383.044,Z 270.395,A -85,B 0,C 180,E1 -12088.493,E2 -12088.493} C_VEL
LIN {X 0,Y 383.006,Z 270.374,A -85,B 0,C 180,E1 -12092.15,E2 -12092.15} C_VEL
LIN {X 0,Y 383.014,Z 270.369,A -85,B 0,C 180,E1 -12094.669,E2 -12094.669} C_VEL
LIN {X 0,Y 382.999,Z 270.401,A -85,B 0,C 180,E1 -12097.905,E2 -12097.905} C_VEL
LIN {X 0,Y 382.999,Z 270.371,A -85,B 0,C 180,E1 -12101.346,E2 -12101.346} C_VEL
LIN {X 0,Y 382.994,Z 270.4,A -85,B 0,C 180,E1 -12104.304,E2 -12104.304} C_VEL
LIN {X 0,Y 383.008,Z 270.38,A -85,B 0,C 180,E1 -12107.241,E2 -12107.241} C_VEL
LIN {X 0,Y 383.014,Z 270.403,A -85,B 0,C 180,E1 -12110.414,E2 -12110.414} C_VEL
LIN {X 0,Y 383.024,Z 270.399,A -85,B 0,C 180,E1 -12114.045,E2 -12114.045} C_VEL
LIN {X 0,Y 382.986,Z 270.405,A -85,B 0,C 180,E1 -12117.579,E2 -12117.579} C_VEL
LIN {X 0,Y 383.066,Z 270.538,A -85,B 0,C 180,E1 -12120.383,E2 -12120.383} C_VEL
LIN {X 0,Y 385.664,Z 281.757,A -85,B 0,C 180,E1 -12123.245,E2 -12123.245} C_VEL
LIN {X 0,Y 386.943,Z 288.126,A -85,B 0,C 180,E1 -12124.726,E2 -12124.726} C_VEL
LIN {X 0,Y 389.979,Z 296.34,A -85,B 0,C 180,E1 -12125.131,E2 -12125.131} C_VEL
LIN {X 0,Y 394.47,Z 318.678,A -85,B 0,C 180,E1 -12125.872,E2 -12125.872} C_VEL
LIN {X 0,Y 392.565,Z 422.052,A -85,B 0,C 180,E1 -12127.779,E2 -12127.779} C_VEL
LIN {X 0,Y 391.974,Z 436.287,A -85,B 0,C 180,E1 -12128.193,E2 -12128.193} C_VEL
LIN {X 0,Y 391.165,Z 450.082,A -85,B 0,C 180,E1 -12128.803,E2 -12128.803} C_VEL
LIN {X 0,Y 390.234,Z 463.187,A -85,B 0,C 180,E1 -12129.593,E2 -12129.593} C_VEL
LIN {X 0,Y 389.089,Z 476.293,A -85,B 0,C 180,E1 -12130.616,E2 -12130.616} C_VEL
LIN {X 0,Y 387.804,Z 488.254,A -85,B 0,C 180,E1 -12131.783,E2 -12131.783} C_VEL
LIN {X 0,Y 386.572,Z 499.164,A -85,B 0,C 180,E1 -12133.089,E2 -12133.089} C_VEL
LIN {X 0,Y 385.243,Z 509.929,A -85,B 0,C 180,E1 -12134.662,E2 -12134.662} C_VEL
LIN {X 0,Y 384.301,Z 518.811,A -85,B 0,C 180,E1 -12136.247,E2 -12136.247} C_VEL
LIN {X 0,Y 383.316,Z 527.316,A -85,B 0,C 180,E1 -12138.097,E2 -12138.097} C_VEL
LIN {X 0,Y 382.614,Z 534.166,A -85,B 0,C 180,E1 -12139.951,E2 -12139.951} C_VEL
LIN {X 0,Y 382.157,Z 538.895,A -85,B 0,C 180,E1 -12141.54,E2 -12141.54} C_VEL
LIN {X 0,Y 381.849,Z 543.793,A -85,B 0,C 180,E1 -12143.66,E2 -12143.66} C_VEL
LIN {X 0,Y 381.647,Z 547.203,A -85,B 0,C 180,E1 -12145.776,E2 -12145.776} C_VEL
LIN {X 0,Y 381.558,Z 549.229,A -85,B 0,C 180,E1 -12147.889,E2 -12147.889} C_VEL
LIN {X 0,Y 381.572,Z 549.924,A -85,B 0,C 180,E1 -12150,E2 -12150} C_VEL
LIN {X 0,Y 381.557,Z 549.298,A -85,B 0,C 180,E1 -12152.111,E2 -12152.111} C_VEL
LIN {X 0,Y 381.647,Z 547.335,A -85,B 0,C 180,E1 -12154.224,E2 -12154.224} C_VEL
LIN {X 0,Y 381.849,Z 543.988,A -85,B 0,C 180,E1 -12156.34,E2 -12156.34} C_VEL
LIN {X 0,Y 382.02,Z 540.904,A -85,B 0,C 180,E1 -12157.77,E2 -12157.77} C_VEL
LIN {X 0,Y 381.508,Z 538.886,A -85,B 0,C 180,E1 -12158.601,E2 -12158.601} C_VEL
LIN {X 0,Y 378.94,Z 535.251,A -85,B 0,C 180,E1 -12159.941,E2 -12159.941} C_VEL
LIN {X 0,Y 376.53,Z 531.048,A -85,B 0,C 180,E1 -12161.257,E2 -12161.257} C_VEL
LIN {X 0,Y 376.268,Z 528.14,A -85,B 0,C 180,E1 -12162.04,E2 -12162.04} C_VEL
LIN {X 0,Y 377.171,Z 520.724,A -85,B 0,C 180,E1 -12163.743,E2 -12163.743} C_VEL
LIN {X 0,Y 378.162,Z 512.212,A -85,B 0,C 180,E1 -12165.356,E2 -12165.356} C_VEL
LIN {X 0,Y 379.446,Z 501.894,A -85,B 0,C 180,E1 -12166.96,E2 -12166.96} C_VEL
LIN {X 0,Y 380.657,Z 491.524,A -85,B 0,C 180,E1 -12168.292,E2 -12168.292} C_VEL
LIN {X 0,Y 381.998,Z 480.245,A -85,B 0,C 180,E1 -12169.479,E2 -12169.479} C_VEL
LIN {X 0,Y 383.192,Z 467.989,A -85,B 0,C 180,E1 -12170.528,E2 -12170.528} C_VEL
LIN {X 0,Y 384.229,Z 455.188,A -85,B 0,C 180,E1 -12171.395,E2 -12171.395} C_VEL
LIN {X 0,Y 385.154,Z 441.15,A -85,B 0,C 180,E1 -12172.107,E2 -12172.107} C_VEL
LIN {X 0,Y 385.865,Z 427.212,A -85,B 0,C 180,E1 -12172.593,E2 -12172.593} C_VEL
LIN {X 0,Y 386.505,Z 403.006,A -85,B 0,C 180,E1 -12173.083,E2 -12173.083} C_VEL
LIN {X 0,Y 387.99,Z 319.148,A -85,B 0,C 180,E1 -12174.653,E2 -12174.653} C_VEL
LIN {X 0,Y 383.439,Z 297.314,A -85,B 0,C 180,E1 -12175.408,E2 -12175.408} C_VEL
LIN {X 0,Y 379.756,Z 288.217,A -85,B 0,C 180,E1 -12175.889,E2 -12175.889} C_VEL
LIN {X 0,Y 377.665,Z 278.304,A -85,B 0,C 180,E1 -12178.307,E2 -12178.307} C_VEL
LIN {X 0,Y 376.028,Z 271.406,A -85,B 0,C 180,E1 -12180.151,E2 -12180.151} C_VEL
LIN {X 0,Y 375.958,Z 271.271,A -85,B 0,C 180,E1 -12184.111,E2 -12184.111} C_VEL
LIN {X 0,Y 375.952,Z 271.278,A -85,B 0,C 180,E1 -12186.74,E2 -12186.74} C_VEL
LIN {X 0,Y 375.987,Z 271.277,A -85,B 0,C 180,E1 -12189.97,E2 -12189.97} C_VEL
LIN {X 0,Y 375.928,Z 271.273,A -85,B 0,C 180,E1 -12193.765,E2 -12193.765} C_VEL
LIN {X 0,Y 375.931,Z 271.271,A -85,B 0,C 180,E1 -12196.81,E2 -12196.81} C_VEL
LIN {X 0,Y 375.964,Z 271.27,A -85,B 0,C 180,E1 -12200.537,E2 -12200.537} C_VEL
LIN {X 0,Y 375.96,Z 271.276,A -85,B 0,C 180,E1 -12203.494,E2 -12203.494} C_VEL
LIN {X 0,Y 375.954,Z 271.246,A -85,B 0,C 180,E1 -12205.888,E2 -12205.888} C_VEL
LIN {X 0,Y 375.962,Z 271.276,A -85,B 0,C 180,E1 -12209.687,E2 -12209.687} C_VEL
LIN {X 0,Y 375.996,Z 271.273,A -85,B 0,C 180,E1 -12212.141,E2 -12212.141} C_VEL
LIN {X 0,Y 376,Z 271.263,A -85,B 0,C 180,E1 -12214.538,E2 -12214.538} C_VEL
LIN {X 0,Y 375.956,Z 271.274,A -85,B 0,C 180,E1 -12218.045,E2 -12218.045} C_VEL
LIN {X 0,Y 376.002,Z 271.273,A -85,B 0,C 180,E1 -12221.473,E2 -12221.473} C_VEL
LIN {X 0,Y 376.051,Z 271.255,A -85,B 0,C 180,E1 -12224.832,E2 -12224.832} C_VEL
LIN {X 0,Y 376.043,Z 271.267,A -85,B 0,C 180,E1 -12228.136,E2 -12228.136} C_VEL
LIN {X 0,Y 376.213,Z 271.234,A -85,B 0,C 180,E1 -12231.917,E2 -12231.917} C_VEL
LIN {X 0,Y 376.165,Z 271.255,A -85,B 0,C 180,E1 -12234.64,E2 -12234.64} C_VEL
LIN {X 0,Y 376.346,Z 271.212,A -85,B 0,C 180,E1 -12237.859,E2 -12237.859} C_VEL
LIN {X 0,Y 376.482,Z 271.21,A -85,B 0,C 180,E1 -12240,E2 -12240} C_VEL
LIN {X 0,Y 376.182,Z 271.237,A -85,B 0,C 180,E1 -12243.213,E2 -12243.213} C_VEL
LIN {X 0,Y 376.238,Z 271.243,A -85,B 0,C 180,E1 -12246.435,E2 -12246.435} C_VEL
LIN {X 0,Y 376.197,Z 271.243,A -85,B 0,C 180,E1 -12248.595,E2 -12248.595} C_VEL
LIN {X 0,Y 376.041,Z 271.261,A -85,B 0,C 180,E1 -12251.864,E2 -12251.864} C_VEL
LIN {X 0,Y 376.05,Z 271.26,A -85,B 0,C 180,E1 -12255.168,E2 -12255.168} C_VEL
LIN {X 0,Y 376.016,Z 271.273,A -85,B 0,C 180,E1 -12258.526,E2 -12258.526} C_VEL
LIN {X 0,Y 375.956,Z 271.269,A -85,B 0,C 180,E1 -12261.955,E2 -12261.955} C_VEL
LIN {X 0,Y 376,Z 271.273,A -85,B 0,C 180,E1 -12265.461,E2 -12265.461} C_VEL
LIN {X 0,Y 375.97,Z 271.274,A -85,B 0,C 180,E1 -12269.079,E2 -12269.079} C_VEL
LIN {X 0,Y 375.944,Z 271.259,A -85,B 0,C 180,E1 -12272.829,E2 -12272.829} C_VEL
LIN {X 0,Y 375.952,Z 271.248,A -85,B 0,C 180,E1 -12275.416,E2 -12275.416} C_VEL
LIN {X 0,Y 375.971,Z 271.278,A -85,B 0,C 180,E1 -12278.271,E2 -12278.271} C_VEL
LIN {X 0,Y 375.93,Z 271.28,A -85,B 0,C 180,E1 -12281.601,E2 -12281.601} C_VEL
LIN {X 0,Y 375.974,Z 271.276,A -85,B 0,C 180,E1 -12285.261,E2 -12285.261} C_VEL
LIN {X 0,Y 375.986,Z 271.254,A -85,B 0,C 180,E1 -12288.39,E2 -12288.39} C_VEL
LIN {X 0,Y 375.965,Z 271.27,A -85,B 0,C 180,E1 -12291.913,E2 -12291.913} C_VEL
LIN {X 0,Y 375.977,Z 271.273,A -85,B 0,C 180,E1 -12295.333,E2 -12295.333} C_VEL
LIN {X 0,Y 375.993,Z 271.449,A -85,B 0,C 180,E1 -12298.671,E2 -12298.671} C_VEL
LIN {X 0,Y 378.932,Z 283.757,A -85,B 0,C 180,E1 -12301.775,E2 -12301.775} C_VEL
LIN {X 0,Y 381.081,Z 294.309,A -85,B 0,C 180,E1 -12304.236,E2 -12304.236} C_VEL
LIN {X 0,Y 382.337,Z 299.716,A -85,B 0,C 180,E1 -12304.475,E2 -12304.475} C_VEL
LIN {X 0,Y 387.814,Z 327.548,A -85,B 0,C 180,E1 -12305.416,E2 -12305.416} C_VEL
LIN {X 0,Y 386.063,Z 425.237,A -85,B 0,C 180,E1 -12307.243,E2 -12307.243} C_VEL
LIN {X 0,Y 385.489,Z 439.97,A -85,B 0,C 180,E1 -12307.631,E2 -12307.631} C_VEL
LIN {X 0,Y 384.599,Z 454.024,A -85,B 0,C 180,E1 -12308.212,E2 -12308.212} C_VEL
LIN {X 0,Y 383.52,Z 468.026,A -85,B 0,C 180,E1 -12309.024,E2 -12309.024} C_VEL
LIN {X 0,Y 382.39,Z 480.659,A -85,B 0,C 180,E1 -12309.983,E2 -12309.983} C_VEL
LIN {X 0,Y 381.028,Z 493.159,A -85,B 0,C 180,E1 -12311.169,E2 -12311.169} C_VEL
LIN {X 0,Y 379.625,Z 504.46,A -85,B 0,C 180,E1 -12312.493,E2 -12312.493} C_VEL
LIN {X 0,Y 378.311,Z 515.529,A -85,B 0,C 180,E1 -12314.097,E2 -12314.097} C_VEL
LIN {X 0,Y 377.321,Z 524.076,A -85,B 0,C 180,E1 -12315.593,E2 -12315.593} C_VEL
LIN {X 0,Y 376.432,Z 532.273,A -85,B 0,C 180,E1 -12317.328,E2 -12317.328} C_VEL
LIN {X 0,Y 375.528,Z 539.535,A -85,B 0,C 180,E1 -12319.214,E2 -12319.214} C_VEL
LIN {X 0,Y 374.979,Z 546.063,A -85,B 0,C 180,E1 -12321.377,E2 -12321.377} C_VEL
LIN {X 0,Y 374.677,Z 550.948,A -85,B 0,C 180,E1 -12323.538,E2 -12323.538} C_VEL
LIN {X 0,Y 374.513,Z 554.344,A -85,B 0,C 180,E1 -12325.695,E2 -12325.695} C_VEL
LIN {X 0,Y 374.41,Z 556.352,A -85,B 0,C 180,E1 -12327.849,E2 -12327.849} C_VEL
LIN {X 0,Y 374.472,Z 557.016,A -85,B 0,C 180,E1 -12330,E2 -12330} C_VEL
LIN {X 0,Y 374.411,Z 556.346,A -85,B 0,C 180,E1 -12332.152,E2 -12332.152} C_VEL
LIN {X 0,Y 374.514,Z 554.335,A -85,B 0,C 180,E1 -12334.305,E2 -12334.305} C_VEL
LIN {X 0,Y 374.677,Z 550.932,A -85,B 0,C 180,E1 -12336.462,E2 -12336.462} C_VEL
LIN {X 0,Y 374.98,Z 546.035,A -85,B 0,C 180,E1 -12338.623,E2 -12338.623} C_VEL
LIN {X 0,Y 375.529,Z 539.501,A -85,B 0,C 180,E1 -12340.786,E2 -12340.786} C_VEL
LIN {X 0,Y 376.437,Z 532.231,A -85,B 0,C 180,E1 -12342.672,E2 -12342.672} C_VEL
LIN {X 0,Y 377.369,Z 523.231,A -85,B 0,C 180,E1 -12344.56,E2 -12344.56} C_VEL
LIN {X 0,Y 378.508,Z 513.772,A -85,B 0,C 180,E1 -12346.171,E2 -12346.171} C_VEL
LIN {X 0,Y 379.766,Z 503.308,A -85,B 0,C 180,E1 -12347.64,E2 -12347.64} C_VEL
LIN {X 0,Y 381.207,Z 491.761,A -85,B 0,C 180,E1 -12348.961,E2 -12348.961} C_VEL
LIN {X 0,Y 382.531,Z 478.948,A -85,B 0,C 180,E1 -12350.15,E2 -12350.15} C_VEL
LIN {X 0,Y 383.743,Z 465.728,A -85,B 0,C 180,E1 -12351.113,E2 -12351.113} C_VEL
LIN {X 0,Y 384.722,Z 452.489,A -85,B 0,C 180,E1 -12351.851,E2 -12351.851} C_VEL
LIN {X 0,Y 385.508,Z 438.734,A -85,B 0,C 180,E1 -12352.403,E2 -12352.403} C_VEL
LIN {X 0,Y 386.061,Z 424.674,A -85,B 0,C 180,E1 -12352.758,E2 -12352.758} C_VEL
LIN {X 0,Y 387.792,Z 327.376,A -85,B 0,C 180,E1 -12354.576,E2 -12354.576} C_VEL
LIN {X 0,Y 381.715,Z 296.67,A -85,B 0,C 180,E1 -12355.618,E2 -12355.618} C_VEL
LIN {X 0,Y 381.059,Z 294.271,A -85,B 0,C 180,E1 -12355.758,E2 -12355.758} C_VEL
LIN {X 0,Y 378.915,Z 283.683,A -85,B 0,C 180,E1 -12358.226,E2 -12358.226} C_VEL
LIN {X 0,Y 375.993,Z 271.418,A -85,B 0,C 180,E1 -12361.327,E2 -12361.327} C_VEL
LIN {X 0,Y 375.978,Z 271.274,A -85,B 0,C 180,E1 -12364.667,E2 -12364.667} C_VEL
LIN {X 0,Y 375.971,Z 271.272,A -85,B 0,C 180,E1 -12368.27,E2 -12368.27} C_VEL
LIN {X 0,Y 375.931,Z 271.26,A -85,B 0,C 180,E1 -12371.6,E2 -12371.6} C_VEL
LIN {X 0,Y 375.924,Z 271.279,A -85,B 0,C 180,E1 -12375.268,E2 -12375.268} C_VEL
LIN {X 0,Y 375.93,Z 271.279,A -85,B 0,C 180,E1 -12378.399,E2 -12378.399} C_VEL
LIN {X 0,Y 375.971,Z 271.278,A -85,B 0,C 180,E1 -12381.729,E2 -12381.729} C_VEL
LIN {X 0,Y 375.975,Z 271.237,A -85,B 0,C 180,E1 -12385.332,E2 -12385.332} C_VEL
LIN {X 0,Y 375.956,Z 271.273,A -85,B 0,C 180,E1 -12388.438,E2 -12388.438} C_VEL
LIN {X 0,Y 375.996,Z 271.265,A -85,B 0,C 180,E1 -12392.141,E2 -12392.141} C_VEL
LIN {X 0,Y 376,Z 271.273,A -85,B 0,C 180,E1 -12394.539,E2 -12394.539} C_VEL
LIN {X 0,Y 375.956,Z 271.269,A -85,B 0,C 180,E1 -12398.045,E2 -12398.045} C_VEL
LIN {X 0,Y 376.017,Z 271.272,A -85,B 0,C 180,E1 -12401.474,E2 -12401.474} C_VEL
LIN {X 0,Y 376.051,Z 271.26,A -85,B 0,C 180,E1 -12404.832,E2 -12404.832} C_VEL
LIN {X 0,Y 376.042,Z 271.261,A -85,B 0,C 180,E1 -12408.136,E2 -12408.136} C_VEL
LIN {X 0,Y 376.25,Z 271.243,A -85,B 0,C 180,E1 -12411.878,E2 -12411.878} C_VEL
LIN {X 0,Y 376.164,Z 271.245,A -85,B 0,C 180,E1 -12414.64,E2 -12414.64} C_VEL
LIN {X 0,Y 376.346,Z 271.229,A -85,B 0,C 180,E1 -12417.86,E2 -12417.86} C_VEL
LIN {X 0,Y 376.481,Z 271.21,A -85,B 0,C 180,E1 -12420,E2 -12420} C_VEL
LIN {X 0,Y 376.183,Z 271.236,A -85,B 0,C 180,E1 -12423.213,E2 -12423.213} C_VEL
LIN {X 0,Y 376.22,Z 271.241,A -85,B 0,C 180,E1 -12426.62,E2 -12426.62} C_VEL
LIN {X 0,Y 376.112,Z 271.25,A -85,B 0,C 180,E1 -12429.682,E2 -12429.682} C_VEL
LIN {X 0,Y 376.083,Z 271.255,A -85,B 0,C 180,E1 -12433.658,E2 -12433.658} C_VEL
LIN {X 0,Y 376.037,Z 271.269,A -85,B 0,C 180,E1 -12437.607,E2 -12437.607} C_VEL
LIN {X 0,Y 375.972,Z 271.266,A -85,B 0,C 180,E1 -12440.833,E2 -12440.833} C_VEL
LIN {X 0,Y 375.988,Z 271.273,A -85,B 0,C 180,E1 -12444.282,E2 -12444.282} C_VEL
LIN {X 0,Y 376.014,Z 271.261,A -85,B 0,C 180,E1 -12446.653,E2 -12446.653} C_VEL
LIN {X 0,Y 375.971,Z 271.279,A -85,B 0,C 180,E1 -12449.079,E2 -12449.079} C_VEL
LIN {X 0,Y 375.945,Z 271.243,A -85,B 0,C 180,E1 -12452.829,E2 -12452.829} C_VEL
LIN {X 0,Y 375.954,Z 271.26,A -85,B 0,C 180,E1 -12455.416,E2 -12455.416} C_VEL
LIN {X 0,Y 375.974,Z 271.277,A -85,B 0,C 180,E1 -12458.272,E2 -12458.272} C_VEL
LIN {X 0,Y 375.945,Z 271.249,A -85,B 0,C 180,E1 -12461.604,E2 -12461.604} C_VEL
LIN {X 0,Y 375.951,Z 271.278,A -85,B 0,C 180,E1 -12465.265,E2 -12465.265} C_VEL
LIN {X 0,Y 375.939,Z 271.275,A -85,B 0,C 180,E1 -12469.134,E2 -12469.134} C_VEL
LIN {X 0,Y 375.963,Z 271.267,A -85,B 0,C 180,E1 -12471.912,E2 -12471.912} C_VEL
LIN {X 0,Y 375.979,Z 271.269,A -85,B 0,C 180,E1 -12475.333,E2 -12475.333} C_VEL
LIN {X 0,Y 375.957,Z 271.273,A -85,B 0,C 180,E1 -12478.439,E2 -12478.439} C_VEL
LIN {X 0,Y 376.02,Z 271.505,A -85,B 0,C 180,E1 -12480.003,E2 -12480.003} C_VEL
LIN {X 0,Y 378.695,Z 282.95,A -85,B 0,C 180,E1 -12482.975,E2 -12482.975} C_VEL
LIN {X 0,Y 379.757,Z 288.146,A -85,B 0,C 180,E1 -12484.208,E2 -12484.208} C_VEL
LIN {X 0,Y 383.812,Z 298.691,A -85,B 0,C 180,E1 -12484.749,E2 -12484.749} C_VEL
LIN {X 0,Y 388.009,Z 320.115,A -85,B 0,C 180,E1 -12485.471,E2 -12485.471} C_VEL
LIN {X 0,Y 385.956,Z 425.043,A -85,B 0,C 180,E1 -12487.448,E2 -12487.448} C_VEL
LIN {X 0,Y 385.277,Z 438.933,A -85,B 0,C 180,E1 -12487.9,E2 -12487.9} C_VEL
LIN {X 0,Y 384.471,Z 451.401,A -85,B 0,C 180,E1 -12488.486,E2 -12488.486} C_VEL
LIN {X 0,Y 383.455,Z 464.958,A -85,B 0,C 180,E1 -12489.347,E2 -12489.347} C_VEL
LIN {X 0,Y 382.214,Z 477.789,A -85,B 0,C 180,E1 -12490.393,E2 -12490.393} C_VEL
LIN {X 0,Y 380.902,Z 489.497,A -85,B 0,C 180,E1 -12491.581,E2 -12491.581} C_VEL
LIN {X 0,Y 379.528,Z 501.182,A -85,B 0,C 180,E1 -12493.043,E2 -12493.043} C_VEL
LIN {X 0,Y 378.188,Z 511.622,A -85,B 0,C 180,E1 -12494.644,E2 -12494.644} C_VEL
LIN {X 0,Y 377.261,Z 520.231,A -85,B 0,C 180,E1 -12496.26,E2 -12496.26} C_VEL
LIN {X 0,Y 376.196,Z 528.485,A -85,B 0,C 180,E1 -12498.141,E2 -12498.141} C_VEL
LIN {X 0,Y 375.601,Z 534.235,A -85,B 0,C 180,E1 -12499.761,E2 -12499.761} C_VEL
LIN {X 0,Y 375.121,Z 538.963,A -85,B 0,C 180,E1 -12501.38,E2 -12501.38} C_VEL
LIN {X 0,Y 374.782,Z 543.861,A -85,B 0,C 180,E1 -12503.54,E2 -12503.54} C_VEL
LIN {X 0,Y 374.579,Z 547.27,A -85,B 0,C 180,E1 -12505.696,E2 -12505.696} C_VEL
LIN {X 0,Y 374.457,Z 549.296,A -85,B 0,C 180,E1 -12507.849,E2 -12507.849} C_VEL
LIN {X 0,Y 374.473,Z 549.991,A -85,B 0,C 180,E1 -12510,E2 -12510} C_VEL
LIN {X 0,Y 374.456,Z 549.364,A -85,B 0,C 180,E1 -12512.151,E2 -12512.151} C_VEL
LIN {X 0,Y 374.579,Z 547.4,A -85,B 0,C 180,E1 -12514.304,E2 -12514.304} C_VEL
LIN {X 0,Y 374.782,Z 544.054,A -85,B 0,C 180,E1 -12516.46,E2 -12516.46} C_VEL
LIN {X 0,Y 375.114,Z 539.227,A -85,B 0,C 180,E1 -12518.62,E2 -12518.62} C_VEL
LIN {X 0,Y 375.776,Z 532.764,A -85,B 0,C 180,E1 -12520.779,E2 -12520.779} C_VEL
LIN {X 0,Y 376.268,Z 528.14,A -85,B 0,C 180,E1 -12522.04,E2 -12522.04} C_VEL
LIN {X 0,Y 376.051,Z 525.078,A -85,B 0,C 180,E1 -12522.809,E2 -12522.809} C_VEL
LIN {X 0,Y 373.89,Z 519.893,A -85,B 0,C 180,E1 -12524.058,E2 -12524.058} C_VEL
LIN {X 0,Y 371.727,Z 514.225,A -85,B 0,C 180,E1 -12525.268,E2 -12525.268} C_VEL
LIN {X 0,Y 371.508,Z 510.402,A -85,B 0,C 180,E1 -12525.964,E2 -12525.964} C_VEL
LIN {X 0,Y 372.857,Z 500.01,A -85,B 0,C 180,E1 -12527.552,E2 -12527.552} C_VEL
LIN {X 0,Y 374.253,Z 489.241,A -85,B 0,C 180,E1 -12528.9,E2 -12528.9} C_VEL
LIN {X 0,Y 375.574,Z 477.459,A -85,B 0,C 180,E1 -12530.111,E2 -12530.111} C_VEL
LIN {X 0,Y 376.86,Z 464.455,A -85,B 0,C 180,E1 -12531.181,E2 -12531.181} C_VEL
LIN {X 0,Y 377.968,Z 450.809,A -85,B 0,C 180,E1 -12532.047,E2 -12532.047} C_VEL
LIN {X 0,Y 378.824,Z 437.251,A -85,B 0,C 180,E1 -12532.676,E2 -12532.676} C_VEL
LIN {X 0,Y 379.45,Z 423.531,A -85,B 0,C 180,E1 -12533.105,E2 -12533.105} C_VEL
LIN {X 0,Y 381.091,Z 345.605,A -85,B 0,C 180,E1 -12534.592,E2 -12534.592} C_VEL
LIN {X 0,Y 381.419,Z 319.646,A -85,B 0,C 180,E1 -12535.097,E2 -12535.097} C_VEL
LIN {X 0,Y 377.318,Z 299.999,A -85,B 0,C 180,E1 -12535.796,E2 -12535.796} C_VEL
LIN {X 0,Y 372.618,Z 288.331,A -85,B 0,C 180,E1 -12536.42,E2 -12536.42} C_VEL
LIN {X 0,Y 371.483,Z 283.1,A -85,B 0,C 180,E1 -12537.683,E2 -12537.683} C_VEL
LIN {X 0,Y 368.951,Z 272.358,A -85,B 0,C 180,E1 -12540.554,E2 -12540.554} C_VEL
LIN {X 0,Y 368.895,Z 272.153,A -85,B 0,C 180,E1 -12543.537,E2 -12543.537} C_VEL
LIN {X 0,Y 368.899,Z 272.154,A -85,B 0,C 180,E1 -12546.855,E2 -12546.855} C_VEL
LIN {X 0,Y 368.909,Z 272.157,A -85,B 0,C 180,E1 -12550.369,E2 -12550.369} C_VEL
LIN {X 0,Y 368.88,Z 272.148,A -85,B 0,C 180,E1 -12553.615,E2 -12553.615} C_VEL
LIN {X 0,Y 368.882,Z 272.151,A -85,B 0,C 180,E1 -12556.695,E2 -12556.695} C_VEL
LIN {X 0,Y 368.931,Z 272.131,A -85,B 0,C 180,E1 -12559.638,E2 -12559.638} C_VEL
LIN {X 0,Y 368.899,Z 272.16,A -85,B 0,C 180,E1 -12563.143,E2 -12563.143} C_VEL
LIN {X 0,Y 368.891,Z 272.12,A -85,B 0,C 180,E1 -12566.461,E2 -12566.461} C_VEL
LIN {X 0,Y 368.917,Z 272.153,A -85,B 0,C 180,E1 -12570.31,E2 -12570.31} C_VEL
LIN {X 0,Y 368.975,Z 272.137,A -85,B 0,C 180,E1 -12573.535,E2 -12573.535} C_VEL
LIN {X 0,Y 368.96,Z 272.15,A -85,B 0,C 180,E1 -12576.421,E2 -12576.421} C_VEL
LIN {X 0,Y 368.929,Z 272.144,A -85,B 0,C 180,E1 -12579.947,E2 -12579.947} C_VEL
LIN {X 0,Y 368.968,Z 272.143,A -85,B 0,C 180,E1 -12583.398,E2 -12583.398} C_VEL
LIN {X 0,Y 369.05,Z 272.135,A -85,B 0,C 180,E1 -12586.79,E2 -12586.79} C_VEL
LIN {X 0,Y 369.06,Z 272.131,A -85,B 0,C 180,E1 -12590.131,E2 -12590.131} C_VEL
LIN {X 0,Y 369.195,Z 272.119,A -85,B 0,C 180,E1 -12593.441,E2 -12593.441} C_VEL
LIN {X 0,Y 369.311,Z 272.088,A -85,B 0,C 180,E1 -12597.819,E2 -12597.819} C_VEL
LIN {X 0,Y 369.452,Z 272.086,A -85,B 0,C 180,E1 -12600,E2 -12600} C_VEL
LIN {X 0,Y 369.311,Z 272.104,A -85,B 0,C 180,E1 -12602.181,E2 -12602.181} C_VEL
LIN {X 0,Y 369.2,Z 272.122,A -85,B 0,C 180,E1 -12606.558,E2 -12606.558} C_VEL
LIN {X 0,Y 369.13,Z 272.122,A -85,B 0,C 180,E1 -12608.761,E2 -12608.761} C_VEL
LIN {X 0,Y 368.997,Z 272.14,A -85,B 0,C 180,E1 -12612.093,E2 -12612.093} C_VEL
LIN {X 0,Y 368.99,Z 272.14,A -85,B 0,C 180,E1 -12615.465,E2 -12615.465} C_VEL
LIN {X 0,Y 368.959,Z 272.149,A -85,B 0,C 180,E1 -12618.894,E2 -12618.894} C_VEL
LIN {X 0,Y 368.925,Z 272.144,A -85,B 0,C 180,E1 -12622.396,E2 -12622.396} C_VEL
LIN {X 0,Y 368.993,Z 272.143,A -85,B 0,C 180,E1 -12625.981,E2 -12625.981} C_VEL
LIN {X 0,Y 368.961,Z 272.148,A -85,B 0,C 180,E1 -12628.814,E2 -12628.814} C_VEL
LIN {X 0,Y 368.894,Z 272.142,A -85,B 0,C 180,E1 -12632.238,E2 -12632.238} C_VEL
LIN {X 0,Y 368.923,Z 272.118,A -85,B 0,C 180,E1 -12635.002,E2 -12635.002} C_VEL
LIN {X 0,Y 368.905,Z 272.156,A -85,B 0,C 180,E1 -12638.641,E2 -12638.641} C_VEL
LIN {X 0,Y 368.877,Z 272.163,A -85,B 0,C 180,E1 -12642.01,E2 -12642.01} C_VEL
LIN {X 0,Y 368.949,Z 272.151,A -85,B 0,C 180,E1 -12645.188,E2 -12645.188} C_VEL
LIN {X 0,Y 368.937,Z 272.131,A -85,B 0,C 180,E1 -12648.186,E2 -12648.186} C_VEL
LIN {X 0,Y 368.911,Z 272.155,A -85,B 0,C 180,E1 -12651.359,E2 -12651.359} C_VEL
LIN {X 0,Y 368.934,Z 272.153,A -85,B 0,C 180,E1 -12655.147,E2 -12655.147} C_VEL
LIN {X 0,Y 368.956,Z 272.363,A -85,B 0,C 180,E1 -12658.243,E2 -12658.243} C_VEL
LIN {X 0,Y 371.666,Z 283.689,A -85,B 0,C 180,E1 -12661.172,E2 -12661.172} C_VEL
LIN {X 0,Y 373.927,Z 294.209,A -85,B 0,C 180,E1 -12663.703,E2 -12663.703} C_VEL
LIN {X 0,Y 375.632,Z 299.485,A -85,B 0,C 180,E1 -12663.982,E2 -12663.982} C_VEL
LIN {X 0,Y 381.386,Z 328.46,A -85,B 0,C 180,E1 -12664.993,E2 -12664.993} C_VEL
LIN {X 0,Y 379.546,Z 425.188,A -85,B 0,C 180,E1 -12666.829,E2 -12666.829} C_VEL
LIN {X 0,Y 378.956,Z 439.914,A -85,B 0,C 180,E1 -12667.224,E2 -12667.224} C_VEL
LIN {X 0,Y 378.011,Z 453.964,A -85,B 0,C 180,E1 -12667.812,E2 -12667.812} C_VEL
LIN {X 0,Y 377.028,Z 466.546,A -85,B 0,C 180,E1 -12668.543,E2 -12668.543} C_VEL
LIN {X 0,Y 375.883,Z 479.014,A -85,B 0,C 180,E1 -12669.478,E2 -12669.478} C_VEL
LIN {X 0,Y 374.427,Z 491.803,A -85,B 0,C 180,E1 -12670.682,E2 -12670.682} C_VEL
LIN {X 0,Y 373.009,Z 503.332,A -85,B 0,C 180,E1 -12672.03,E2 -12672.03} C_VEL
LIN {X 0,Y 371.665,Z 513.778,A -85,B 0,C 180,E1 -12673.523,E2 -12673.523} C_VEL
LIN {X 0,Y 370.49,Z 523.442,A -85,B 0,C 180,E1 -12675.206,E2 -12675.206} C_VEL
LIN {X 0,Y 369.476,Z 532.207,A -85,B 0,C 180,E1 -12677.085,E2 -12677.085} C_VEL
LIN {X 0,Y 368.511,Z 539.469,A -85,B 0,C 180,E1 -12679.006,E2 -12679.006} C_VEL
LIN {X 0,Y 367.917,Z 545.997,A -85,B 0,C 180,E1 -12681.21,E2 -12681.21} C_VEL
LIN {X 0,Y 367.588,Z 550.882,A -85,B 0,C 180,E1 -12683.413,E2 -12683.413} C_VEL
LIN {X 0,Y 367.423,Z 554.278,A -85,B 0,C 180,E1 -12685.612,E2 -12685.612} C_VEL
LIN {X 0,Y 367.314,Z 556.285,A -85,B 0,C 180,E1 -12687.807,E2 -12687.807} C_VEL
LIN {X 0,Y 367.372,Z 556.949,A -85,B 0,C 180,E1 -12690,E2 -12690} C_VEL
LIN {X 0,Y 367.314,Z 556.28,A -85,B 0,C 180,E1 -12692.193,E2 -12692.193} C_VEL
LIN {X 0,Y 367.424,Z 554.268,A -85,B 0,C 180,E1 -12694.388,E2 -12694.388} C_VEL
LIN {X 0,Y 367.587,Z 550.865,A -85,B 0,C 180,E1 -12696.587,E2 -12696.587} C_VEL
LIN {X 0,Y 367.918,Z 545.967,A -85,B 0,C 180,E1 -12698.79,E2 -12698.79} C_VEL
LIN {X 0,Y 368.511,Z 539.432,A -85,B 0,C 180,E1 -12700.994,E2 -12700.994} C_VEL
LIN {X 0,Y 369.478,Z 532.162,A -85,B 0,C 180,E1 -12702.915,E2 -12702.915} C_VEL
LIN {X 0,Y 370.453,Z 523.157,A -85,B 0,C 180,E1 -12704.839,E2 -12704.839} C_VEL
LIN {X 0,Y 371.659,Z 513.702,A -85,B 0,C 180,E1 -12706.478,E2 -12706.478} C_VEL
LIN {X 0,Y 372.991,Z 503.238,A -85,B 0,C 180,E1 -12707.971,E2 -12707.971} C_VEL
LIN {X 0,Y 374.475,Z 491.691,A -85,B 0,C 180,E1 -12709.316,E2 -12709.316} C_VEL
LIN {X 0,Y 375.861,Z 478.876,A -85,B 0,C 180,E1 -12710.523,E2 -12710.523} C_VEL
LIN {X 0,Y 377.067,Z 466.361,A -85,B 0,C 180,E1 -12711.455,E2 -12711.455} C_VEL
LIN {X 0,Y 378.053,Z 453.716,A -85,B 0,C 180,E1 -12712.185,E2 -12712.185} C_VEL
LIN {X 0,Y 378.913,Z 439.572,A -85,B 0,C 180,E1 -12712.779,E2 -12712.779} C_VEL
LIN {X 0,Y 379.486,Z 426.141,A -85,B 0,C 180,E1 -12713.139,E2 -12713.139} C_VEL
LIN {X 0,Y 381.363,Z 328.799,A -85,B 0,C 180,E1 -12714.988,E2 -12714.988} C_VEL
LIN {X 0,Y 375.608,Z 299.223,A -85,B 0,C 180,E1 -12716.011,E2 -12716.011} C_VEL
LIN {X 0,Y 373.887,Z 294.142,A -85,B 0,C 180,E1 -12716.297,E2 -12716.297} C_VEL
LIN {X 0,Y 371.645,Z 283.612,A -85,B 0,C 180,E1 -12718.83,E2 -12718.83} C_VEL
LIN {X 0,Y 368.94,Z 272.319,A -85,B 0,C 180,E1 -12721.757,E2 -12721.757} C_VEL
LIN {X 0,Y 368.927,Z 272.157,A -85,B 0,C 180,E1 -12725.001,E2 -12725.001} C_VEL
LIN {X 0,Y 368.906,Z 272.157,A -85,B 0,C 180,E1 -12728.64,E2 -12728.64} C_VEL
LIN {X 0,Y 368.878,Z 272.14,A -85,B 0,C 180,E1 -12732.009,E2 -12732.009} C_VEL
LIN {X 0,Y 368.877,Z 272.157,A -85,B 0,C 180,E1 -12735.175,E2 -12735.175} C_VEL
LIN {X 0,Y 368.879,Z 272.16,A -85,B 0,C 180,E1 -12738.177,E2 -12738.177} C_VEL
LIN {X 0,Y 368.906,Z 272.156,A -85,B 0,C 180,E1 -12741.359,E2 -12741.359} C_VEL
LIN {X 0,Y 368.932,Z 272.114,A -85,B 0,C 180,E1 -12745.146,E2 -12745.146} C_VEL
LIN {X 0,Y 368.924,Z 272.152,A -85,B 0,C 180,E1 -12749.046,E2 -12749.046} C_VEL
LIN {X 0,Y 368.981,Z 272.143,A -85,B 0,C 180,E1 -12751.564,E2 -12751.564} C_VEL
LIN {X 0,Y 368.952,Z 272.15,A -85,B 0,C 180,E1 -12755.224,E2 -12755.224} C_VEL
LIN {X 0,Y 368.931,Z 272.147,A -85,B 0,C 180,E1 -12758.973,E2 -12758.973} C_VEL
LIN {X 0,Y 368.984,Z 272.139,A -85,B 0,C 180,E1 -12762.257,E2 -12762.257} C_VEL
LIN {X 0,Y 369.03,Z 272.142,A -85,B 0,C 180,E1 -12766.228,E2 -12766.228} C_VEL
LIN {X 0,Y 369.06,Z 272.126,A -85,B 0,C 180,E1 -12770.132,E2 -12770.132} C_VEL
LIN {X 0,Y 369.181,Z 272.121,A -85,B 0,C 180,E1 -12772.342,E2 -12772.342} C_VEL
LIN {X 0,Y 369.137,Z 272.12,A -85,B 0,C 180,E1 -12774.538,E2 -12774.538} C_VEL
LIN {X 0,Y 369.311,Z 272.104,A -85,B 0,C 180,E1 -12777.819,E2 -12777.819} C_VEL
LIN {X 0,Y 369.451,Z 272.086,A -85,B 0,C 180,E1 -12780,E2 -12780} C_VEL
LIN {X 0,Y 369.312,Z 272.088,A -85,B 0,C 180,E1 -12782.181,E2 -12782.181} C_VEL
LIN {X 0,Y 369.19,Z 272.119,A -85,B 0,C 180,E1 -12786.605,E2 -12786.605} C_VEL
LIN {X 0,Y 369.06,Z 272.13,A -85,B 0,C 180,E1 -12789.869,E2 -12789.869} C_VEL
LIN {X 0,Y 369.03,Z 272.132,A -85,B 0,C 180,E1 -12793.772,E2 -12793.772} C_VEL
LIN {X 0,Y 368.995,Z 272.145,A -85,B 0,C 180,E1 -12797.769,E2 -12797.769} C_VEL
LIN {X 0,Y 368.923,Z 272.144,A -85,B 0,C 180,E1 -12801.22,E2 -12801.22} C_VEL
LIN {X 0,Y 368.952,Z 272.15,A -85,B 0,C 180,E1 -12804.776,E2 -12804.776} C_VEL
LIN {X 0,Y 368.982,Z 272.146,A -85,B 0,C 180,E1 -12808.436,E2 -12808.436} C_VEL
LIN {X 0,Y 368.894,Z 272.127,A -85,B 0,C 180,E1 -12812.239,E2 -12812.239} C_VEL
LIN {X 0,Y 368.925,Z 272.127,A -85,B 0,C 180,E1 -12815.002,E2 -12815.002} C_VEL
LIN {X 0,Y 368.909,Z 272.155,A -85,B 0,C 180,E1 -12818.642,E2 -12818.642} C_VEL
LIN {X 0,Y 368.887,Z 272.129,A -85,B 0,C 180,E1 -12822.012,E2 -12822.012} C_VEL
LIN {X 0,Y 368.904,Z 272.157,A -85,B 0,C 180,E1 -12825.181,E2 -12825.181} C_VEL
LIN {X 0,Y 368.881,Z 272.14,A -85,B 0,C 180,E1 -12828.178,E2 -12828.178} C_VEL
LIN {X 0,Y 368.907,Z 272.151,A -85,B 0,C 180,E1 -12831.36,E2 -12831.36} C_VEL
LIN {X 0,Y 368.935,Z 272.148,A -85,B 0,C 180,E1 -12835.147,E2 -12835.147} C_VEL
LIN {X 0,Y 368.929,Z 272.149,A -85,B 0,C 180,E1 -12839.047,E2 -12839.047} C_VEL
LIN {X 0,Y 368.939,Z 272.277,A -85,B 0,C 180,E1 -12839.524,E2 -12839.524} C_VEL
LIN {X 0,Y 371.437,Z 282.693,A -85,B 0,C 180,E1 -12842.323,E2 -12842.323} C_VEL
LIN {X 0,Y 372.572,Z 288.174,A -85,B 0,C 180,E1 -12843.667,E2 -12843.667} C_VEL
LIN {X 0,Y 377.694,Z 301.363,A -85,B 0,C 180,E1 -12844.364,E2 -12844.364} C_VEL
LIN {X 0,Y 381.517,Z 320.307,A -85,B 0,C 180,E1 -12845.027,E2 -12845.027} C_VEL
LIN {X 0,Y 379.773,Z 408.658,A -85,B 0,C 180,E1 -12846.699,E2 -12846.699} C_VEL
LIN {X 0,Y 379.236,Z 428.55,A -85,B 0,C 180,E1 -12847.133,E2 -12847.133} C_VEL
LIN {X 0,Y 378.451,Z 442.816,A -85,B 0,C 180,E1 -12847.66,E2 -12847.66} C_VEL
LIN {X 0,Y 377.484,Z 456.587,A -85,B 0,C 180,E1 -12848.392,E2 -12848.392} C_VEL
LIN {X 0,Y 376.339,Z 470.194,A -85,B 0,C 180,E1 -12849.361,E2 -12849.361} C_VEL
LIN {X 0,Y 375.04,Z 482.075,A -85,B 0,C 180,E1 -12850.43,E2 -12850.43} C_VEL
LIN {X 0,Y 373.574,Z 494.107,A -85,B 0,C 180,E1 -12851.774,E2 -12851.774} C_VEL
LIN {X 0,Y 372.231,Z 504.953,A -85,B 0,C 180,E1 -12853.266,E2 -12853.266} C_VEL
LIN {X 0,Y 370.924,Z 514.801,A -85,B 0,C 180,E1 -12854.915,E2 -12854.915} C_VEL
LIN {X 0,Y 370.059,Z 522.812,A -85,B 0,C 180,E1 -12856.547,E2 -12856.547} C_VEL
LIN {X 0,Y 368.975,Z 530.566,A -85,B 0,C 180,E1 -12858.463,E2 -12858.463} C_VEL
LIN {X 0,Y 368.414,Z 535.981,A -85,B 0,C 180,E1 -12860.114,E2 -12860.114} C_VEL
LIN {X 0,Y 367.848,Z 541.674,A -85,B 0,C 180,E1 -12862.314,E2 -12862.314} C_VEL
LIN {X 0,Y 367.699,Z 544.419,A -85,B 0,C 180,E1 -12863.669,E2 -12863.669} C_VEL
LIN {X 0,Y 367.511,Z 547.338,A -85,B 0,C 180,E1 -12865.613,E2 -12865.613} C_VEL
LIN {X 0,Y 367.358,Z 549.363,A -85,B 0,C 180,E1 -12867.807,E2 -12867.807} C_VEL
LIN {X 0,Y 367.373,Z 550.057,A -85,B 0,C 180,E1 -12870,E2 -12870} C_VEL
LIN {X 0,Y 367.357,Z 549.431,A -85,B 0,C 180,E1 -12872.193,E2 -12872.193} C_VEL
LIN {X 0,Y 367.512,Z 547.466,A -85,B 0,C 180,E1 -12874.387,E2 -12874.387} C_VEL
LIN {X 0,Y 367.728,Z 544.12,A -85,B 0,C 180,E1 -12876.584,E2 -12876.584} C_VEL
LIN {X 0,Y 368.063,Z 539.293,A -85,B 0,C 180,E1 -12878.786,E2 -12878.786} C_VEL
LIN {X 0,Y 368.748,Z 532.829,A -85,B 0,C 180,E1 -12880.987,E2 -12880.987} C_VEL
LIN {X 0,Y 369.652,Z 525.631,A -85,B 0,C 180,E1 -12882.908,E2 -12882.908} C_VEL
LIN {X 0,Y 370.708,Z 516.932,A -85,B 0,C 180,E1 -12884.788,E2 -12884.788} C_VEL
LIN {X 0,Y 371.508,Z 510.402,A -85,B 0,C 180,E1 -12885.964,E2 -12885.964} C_VEL
LIN {X 0,Y 371.346,Z 506.468,A -85,B 0,C 180,E1 -12886.639,E2 -12886.639} C_VEL
LIN {X 0,Y 369.468,Z 499.862,A -85,B 0,C 180,E1 -12887.745,E2 -12887.745} C_VEL
LIN {X 0,Y 367.694,Z 492.9,A -85,B 0,C 180,E1 -12888.803,E2 -12888.803} C_VEL
LIN {X 0,Y 367.661,Z 488.275,A -85,B 0,C 180,E1 -12889.38,E2 -12889.38} C_VEL
LIN {X 0,Y 369.124,Z 476.094,A -85,B 0,C 180,E1 -12890.623,E2 -12890.623} C_VEL
LIN {X 0,Y 370.402,Z 462.799,A -85,B 0,C 180,E1 -12891.702,E2 -12891.702} C_VEL
LIN {X 0,Y 371.467,Z 449.57,A -85,B 0,C 180,E1 -12892.527,E2 -12892.527} C_VEL
LIN {X 0,Y 372.392,Z 435.474,A -85,B 0,C 180,E1 -12893.164,E2 -12893.164} C_VEL
LIN {X 0,Y 372.989,Z 422.072,A -85,B 0,C 180,E1 -12893.566,E2 -12893.566} C_VEL
LIN {X 0,Y 374.659,Z 345.898,A -85,B 0,C 180,E1 -12895.038,E2 -12895.038} C_VEL
LIN {X 0,Y 375.021,Z 320.828,A -85,B 0,C 180,E1 -12895.532,E2 -12895.532} C_VEL
LIN {X 0,Y 371.123,Z 302.328,A -85,B 0,C 180,E1 -12896.211,E2 -12896.211} C_VEL
LIN {X 0,Y 365.365,Z 288.28,A -85,B 0,C 180,E1 -12896.998,E2 -12896.998} C_VEL
LIN {X 0,Y 363.085,Z 277.88,A -85,B 0,C 180,E1 -12899.693,E2 -12899.693} C_VEL
LIN {X 0,Y 361.876,Z 273.094,A -85,B 0,C 180,E1 -12901.091,E2 -12901.091} C_VEL
LIN {X 0,Y 361.853,Z 273.027,A -85,B 0,C 180,E1 -12904.28,E2 -12904.28} C_VEL
LIN {X 0,Y 361.862,Z 273.026,A -85,B 0,C 180,E1 -12907.222,E2 -12907.222} C_VEL
LIN {X 0,Y 361.834,Z 273.036,A -85,B 0,C 180,E1 -12910.755,E2 -12910.755} C_VEL
LIN {X 0,Y 361.818,Z 273.038,A -85,B 0,C 180,E1 -12914.367,E2 -12914.367} C_VEL
LIN {X 0,Y 361.838,Z 273.013,A -85,B 0,C 180,E1 -12917.566,E2 -12917.566} C_VEL
LIN {X 0,Y 361.87,Z 273.028,A -85,B 0,C 180,E1 -12920.972,E2 -12920.972} C_VEL
LIN {X 0,Y 361.87,Z 273.016,A -85,B 0,C 180,E1 -12924.654,E2 -12924.654} C_VEL
LIN {X 0,Y 361.833,Z 273.017,A -85,B 0,C 180,E1 -12928.37,E2 -12928.37} C_VEL
LIN {X 0,Y 361.897,Z 273.033,A -85,B 0,C 180,E1 -12930.955,E2 -12930.955} C_VEL
LIN {X 0,Y 361.949,Z 273.012,A -85,B 0,C 180,E1 -12933.474,E2 -12933.474} C_VEL
LIN {X 0,Y 361.883,Z 273.031,A -85,B 0,C 180,E1 -12937.144,E2 -12937.144} C_VEL
LIN {X 0,Y 361.899,Z 273.024,A -85,B 0,C 180,E1 -12940.723,E2 -12940.723} C_VEL
LIN {X 0,Y 361.925,Z 273.023,A -85,B 0,C 180,E1 -12943.066,E2 -12943.066} C_VEL
LIN {X 0,Y 361.991,Z 273.011,A -85,B 0,C 180,E1 -12946.527,E2 -12946.527} C_VEL
LIN {X 0,Y 362.024,Z 273.008,A -85,B 0,C 180,E1 -12949.938,E2 -12949.938} C_VEL
LIN {X 0,Y 362.157,Z 272.996,A -85,B 0,C 180,E1 -12953.313,E2 -12953.313} C_VEL
LIN {X 0,Y 362.275,Z 272.964,A -85,B 0,C 180,E1 -12957.776,E2 -12957.776} C_VEL
LIN {X 0,Y 362.422,Z 272.961,A -85,B 0,C 180,E1 -12960,E2 -12960} C_VEL
LIN {X 0,Y 362.275,Z 272.98,A -85,B 0,C 180,E1 -12962.224,E2 -12962.224} C_VEL
LIN {X 0,Y 362.164,Z 272.998,A -85,B 0,C 180,E1 -12966.686,E2 -12966.686} C_VEL
LIN {X 0,Y 362.066,Z 273,A -85,B 0,C 180,E1 -12968.933,E2 -12968.933} C_VEL
